LIN {X 0,Y 360.281,Z 704.675,A -85,B 0,C 180,E1 -13053.355,E2 -13053.355} C_VEL
LIN {X 0,Y 360.322,Z 702.646,A -85,B 0,C 180,E1 -13055.597,E2 -13055.597} C_VEL
LIN {X 0,Y 360.498,Z 699.39,A -85,B 0,C 180,E1 -13057.843,E2 -13057.843} C_VEL
LIN {X 0,Y 360.868,Z 694.879,A -85,B 0,C 180,E1 -13060.095,E2 -13060.095} C_VEL
LIN {X 0,Y 361.629,Z 689.019,A -85,B 0,C 180,E1 -13062.344,E2 -13062.344} C_VEL
LIN {X 0,Y 362.564,Z 681.663,A -85,B 0,C 180,E1 -13064.596,E2 -13064.596} C_VEL
LIN {X 0,Y 363.854,Z 673.825,A -85,B 0,C 180,E1 -13066.553,E2 -13066.553} C_VEL
LIN {X 0,Y 365.455,Z 664.444,A -85,B 0,C 180,E1 -13068.5,E2 -13068.5} C_VEL
LIN {X 0,Y 367.139,Z 654.928,A -85,B 0,C 180,E1 -13070.155,E2 -13070.155} C_VEL
LIN {X 0,Y 369.018,Z 643.667,A -85,B 0,C 180,E1 -13071.801,E2 -13071.801} C_VEL
LIN {X 0,Y 371.077,Z 631.324,A -85,B 0,C 180,E1 -13073.289,E2 -13073.289} C_VEL
LIN {X 0,Y 373.236,Z 617.701,A -85,B 0,C 180,E1 -13074.621,E2 -13074.621} C_VEL
LIN {X 0,Y 375.112,Z 604.087,A -85,B 0,C 180,E1 -13075.697,E2 -13075.697} C_VEL
LIN {X 0,Y 376.684,Z 589.68,A -85,B 0,C 180,E1 -13076.601,E2 -13076.601} C_VEL
LIN {X 0,Y 378.096,Z 575.109,A -85,B 0,C 180,E1 -13077.278,E2 -13077.278} C_VEL
LIN {X 0,Y 379.101,Z 560.278,A -85,B 0,C 180,E1 -13077.761,E2 -13077.761} C_VEL
LIN {X 0,Y 380.462,Z 514.951,A -85,B 0,C 180,E1 -13078.666,E2 -13078.666} C_VEL
LIN {X 0,Y 382.505,Z 436.101,A -85,B 0,C 180,E1 -13080.202,E2 -13080.202} C_VEL
LIN {X 0,Y 378.894,Z 417.126,A -85,B 0,C 180,E1 -13080.986,E2 -13080.986} C_VEL
LIN {X 0,Y 377.468,Z 411.276,A -85,B 0,C 180,E1 -13081.265,E2 -13081.265} C_VEL
LIN {X 0,Y 372.216,Z 400.047,A -85,B 0,C 180,E1 -13082.081,E2 -13082.081} C_VEL
LIN {X 0,Y 368.416,Z 392.244,A -85,B 0,C 180,E1 -13082.715,E2 -13082.715} C_VEL
LIN {X 0,Y 365.416,Z 380.947,A -85,B 0,C 180,E1 -13085.538,E2 -13085.538} C_VEL
LIN {X 0,Y 361.841,Z 369.028,A -85,B 0,C 180,E1 -13088.773,E2 -13088.773} C_VEL
LIN {X 0,Y 361.828,Z 369.03,A -85,B 0,C 180,E1 -13092.431,E2 -13092.431} C_VEL
LIN {X 0,Y 361.815,Z 369.04,A -85,B 0,C 180,E1 -13095.947,E2 -13095.947} C_VEL
LIN {X 0,Y 361.811,Z 369.041,A -85,B 0,C 180,E1 -13099.249,E2 -13099.249} C_VEL
LIN {X 0,Y 361.862,Z 369.019,A -85,B 0,C 180,E1 -13102.982,E2 -13102.982} C_VEL
LIN {X 0,Y 361.861,Z 369.033,A -85,B 0,C 180,E1 -13106.63,E2 -13106.63} C_VEL
LIN {X 0,Y 361.864,Z 369.009,A -85,B 0,C 180,E1 -13109.672,E2 -13109.672} C_VEL
LIN {X 0,Y 361.873,Z 369.027,A -85,B 0,C 180,E1 -13113.469,E2 -13113.469} C_VEL
LIN {X 0,Y 361.88,Z 369.026,A -85,B 0,C 180,E1 -13117.144,E2 -13117.144} C_VEL
LIN {X 0,Y 361.888,Z 369.027,A -85,B 0,C 180,E1 -13120.723,E2 -13120.723} C_VEL
LIN {X 0,Y 361.933,Z 369.022,A -85,B 0,C 180,E1 -13123.066,E2 -13123.066} C_VEL
LIN {X 0,Y 362,Z 369.016,A -85,B 0,C 180,E1 -13126.528,E2 -13126.528} C_VEL
LIN {X 0,Y 362.001,Z 369.018,A -85,B 0,C 180,E1 -13129.938,E2 -13129.938} C_VEL
LIN {X 0,Y 362.125,Z 369.001,A -85,B 0,C 180,E1 -13133.313,E2 -13133.313} C_VEL
LIN {X 0,Y 362.278,Z 368.982,A -85,B 0,C 180,E1 -13137.777,E2 -13137.777} C_VEL
LIN {X 0,Y 362.206,Z 368.992,A -85,B 0,C 180,E1 -13141.112,E2 -13141.112} C_VEL
LIN {X 0,Y 362.271,Z 368.984,A -85,B 0,C 180,E1 -13142.224,E2 -13142.224} C_VEL
LIN {X 0,Y 362.126,Z 368.996,A -85,B 0,C 180,E1 -13146.688,E2 -13146.688} C_VEL
LIN {X 0,Y 362.03,Z 369.014,A -85,B 0,C 180,E1 -13150.063,E2 -13150.063} C_VEL
LIN {X 0,Y 362,Z 369.017,A -85,B 0,C 180,E1 -13153.899,E2 -13153.899} C_VEL
LIN {X 0,Y 361.97,Z 369.011,A -85,B 0,C 180,E1 -13157.939,E2 -13157.939} C_VEL
LIN {X 0,Y 361.863,Z 369.029,A -85,B 0,C 180,E1 -13161.655,E2 -13161.655} C_VEL
LIN {X 0,Y 361.872,Z 369.011,A -85,B 0,C 180,E1 -13165.295,E2 -13165.295} C_VEL
LIN {X 0,Y 361.877,Z 369.03,A -85,B 0,C 180,E1 -13169.08,E2 -13169.08} C_VEL
LIN {X 0,Y 361.851,Z 369.038,A -85,B 0,C 180,E1 -13172.945,E2 -13172.945} C_VEL
LIN {X 0,Y 361.867,Z 369.018,A -85,B 0,C 180,E1 -13175.638,E2 -13175.638} C_VEL
LIN {X 0,Y 361.828,Z 369.028,A -85,B 0,C 180,E1 -13179.018,E2 -13179.018} C_VEL
LIN {X 0,Y 361.836,Z 369.03,A -85,B 0,C 180,E1 -13182.83,E2 -13182.83} C_VEL
LIN {X 0,Y 361.874,Z 369.139,A -85,B 0,C 180,E1 -13185.189,E2 -13185.189} C_VEL
LIN {X 0,Y 363.464,Z 374.54,A -85,B 0,C 180,E1 -13186.781,E2 -13186.781} C_VEL
LIN {X 0,Y 374.259,Z 394.401,A -85,B 0,C 180,E1 -13188.479,E2 -13188.479} C_VEL
LIN {X 0,Y 382.475,Z 411.542,A -85,B 0,C 180,E1 -13189.721,E2 -13189.721} C_VEL
LIN {X 0,Y 383.173,Z 413.081,A -85,B 0,C 180,E1 -13189.825,E2 -13189.825} C_VEL
LIN {X 0,Y 379.937,Z 522.43,A -85,B 0,C 180,E1 -13191.918,E2 -13191.918} C_VEL
LIN {X 0,Y 379.375,Z 541.692,A -85,B 0,C 180,E1 -13192.35,E2 -13192.35} C_VEL
LIN {X 0,Y 378.405,Z 556.889,A -85,B 0,C 180,E1 -13192.885,E2 -13192.885} C_VEL
LIN {X 0,Y 377.255,Z 570.714,A -85,B 0,C 180,E1 -13193.572,E2 -13193.572} C_VEL
LIN {X 0,Y 375.754,Z 583.754,A -85,B 0,C 180,E1 -13194.398,E2 -13194.398} C_VEL
LIN {X 0,Y 374.107,Z 597.673,A -85,B 0,C 180,E1 -13195.533,E2 -13195.533} C_VEL
LIN {X 0,Y 372.22,Z 610.378,A -85,B 0,C 180,E1 -13196.8,E2 -13196.8} C_VEL
LIN {X 0,Y 370.129,Z 623.095,A -85,B 0,C 180,E1 -13198.346,E2 -13198.346} C_VEL
LIN {X 0,Y 368.249,Z 633.861,A -85,B 0,C 180,E1 -13199.935,E2 -13199.935} C_VEL
LIN {X 0,Y 366.464,Z 644.127,A -85,B 0,C 180,E1 -13201.755,E2 -13201.755} C_VEL
LIN {X 0,Y 364.771,Z 653.232,A -85,B 0,C 180,E1 -13203.696,E2 -13203.696} C_VEL
LIN {X 0,Y 363.385,Z 660.855,A -85,B 0,C 180,E1 -13205.661,E2 -13205.661} C_VEL
LIN {X 0,Y 362.26,Z 667.561,A -85,B 0,C 180,E1 -13207.771,E2 -13207.771} C_VEL
LIN {X 0,Y 361.372,Z 673.427,A -85,B 0,C 180,E1 -13210.102,E2 -13210.102} C_VEL
LIN {X 0,Y 360.817,Z 678.163,A -85,B 0,C 180,E1 -13212.637,E2 -13212.637} C_VEL
LIN {X 0,Y 360.53,Z 680.275,A -85,B 0,C 180,E1 -13214.163,E2 -13214.163} C_VEL
LIN {X 0,Y 360.307,Z 682.413,A -85,B 0,C 180,E1 -13216.463,E2 -13216.463} C_VEL
LIN {X 0,Y 360.253,Z 683.361,A -85,B 0,C 180,E1 -13218.75,E2 -13218.75} C_VEL
LIN {X 0,Y 360.177,Z 683.159,A -85,B 0,C 180,E1 -13221.019,E2 -13221.019} C_VEL
LIN {X 0,Y 360.356,Z 681.807,A -85,B 0,C 180,E1 -13223.28,E2 -13223.28} C_VEL
LIN {X 0,Y 360.509,Z 679.255,A -85,B 0,C 180,E1 -13225.528,E2 -13225.528} C_VEL
LIN {X 0,Y 360.794,Z 675.491,A -85,B 0,C 180,E1 -13227.767,E2 -13227.767} C_VEL
LIN {X 0,Y 361.121,Z 670.466,A -85,B 0,C 180,E1 -13230,E2 -13230} C_VEL
LIN {X 0,Y 361.852,Z 664.03,A -85,B 0,C 180,E1 -13232.226,E2 -13232.226} C_VEL
LIN {X 0,Y 362.935,Z 655.999,A -85,B 0,C 180,E1 -13234.443,E2 -13234.443} C_VEL
LIN {X 0,Y 364.185,Z 647.445,A -85,B 0,C 180,E1 -13236.371,E2 -13236.371} C_VEL
LIN {X 0,Y 365.609,Z 637.19,A -85,B 0,C 180,E1 -13238.289,E2 -13238.289} C_VEL
LIN {X 0,Y 367.078,Z 626.692,A -85,B 0,C 180,E1 -13239.922,E2 -13239.922} C_VEL
LIN {X 0,Y 368.588,Z 615.282,A -85,B 0,C 180,E1 -13241.41,E2 -13241.41} C_VEL
LIN {X 0,Y 370.142,Z 602.884,A -85,B 0,C 180,E1 -13242.752,E2 -13242.752} C_VEL
LIN {X 0,Y 371.609,Z 590.122,A -85,B 0,C 180,E1 -13243.886,E2 -13243.886} C_VEL
LIN {X 0,Y 371.551,Z 584.912,A -85,B 0,C 180,E1 -13244.323,E2 -13244.323} C_VEL
LIN {X 0,Y 369.644,Z 576.463,A -85,B 0,C 180,E1 -13245.078,E2 -13245.078} C_VEL
LIN {X 0,Y 367.665,Z 567.83,A -85,B 0,C 180,E1 -13245.765,E2 -13245.765} C_VEL
LIN {X 0,Y 367.506,Z 562.338,A -85,B 0,C 180,E1 -13246.09,E2 -13246.09} C_VEL
LIN {X 0,Y 368.412,Z 546.776,A -85,B 0,C 180,E1 -13246.735,E2 -13246.735} C_VEL
LIN {X 0,Y 369.037,Z 531.674,A -85,B 0,C 180,E1 -13247.133,E2 -13247.133} C_VEL
LIN {X 0,Y 371.931,Z 411.976,A -85,B 0,C 180,E1 -13249.45,E2 -13249.45} C_VEL
LIN {X 0,Y 369.611,Z 405.572,A -85,B 0,C 180,E1 -13249.766,E2 -13249.766} C_VEL
LIN {X 0,Y 360.274,Z 383.68,A -85,B 0,C 180,E1 -13251,E2 -13251} C_VEL
LIN {X 0,Y 355.812,Z 373.961,A -85,B 0,C 180,E1 -13251.636,E2 -13251.636} C_VEL
LIN {X 0,Y 354.836,Z 369.91,A -85,B 0,C 180,E1 -13252.72,E2 -13252.72} C_VEL
LIN {X 0,Y 354.807,Z 369.916,A -85,B 0,C 180,E1 -13255.835,E2 -13255.835} C_VEL
LIN {X 0,Y 354.804,Z 369.909,A -85,B 0,C 180,E1 -13259.683,E2 -13259.683} C_VEL
LIN {X 0,Y 354.791,Z 369.907,A -85,B 0,C 180,E1 -13262.333,E2 -13262.333} C_VEL
LIN {X 0,Y 354.825,Z 369.904,A -85,B 0,C 180,E1 -13265.699,E2 -13265.699} C_VEL
LIN {X 0,Y 354.772,Z 369.913,A -85,B 0,C 180,E1 -13269.412,E2 -13269.412} C_VEL
LIN {X 0,Y 354.789,Z 369.914,A -85,B 0,C 180,E1 -13272.866,E2 -13272.866} C_VEL
LIN {X 0,Y 354.769,Z 369.902,A -85,B 0,C 180,E1 -13276.103,E2 -13276.103} C_VEL
LIN {X 0,Y 354.769,Z 369.919,A -85,B 0,C 180,E1 -13279.176,E2 -13279.176} C_VEL
LIN {X 0,Y 354.802,Z 369.912,A -85,B 0,C 180,E1 -13282.404,E2 -13282.404} C_VEL
LIN {X 0,Y 354.811,Z 369.911,A -85,B 0,C 180,E1 -13284.94,E2 -13284.94} C_VEL
LIN {X 0,Y 354.796,Z 369.915,A -85,B 0,C 180,E1 -13288.405,E2 -13288.405} C_VEL
LIN {X 0,Y 354.8,Z 369.891,A -85,B 0,C 180,E1 -13291.614,E2 -13291.614} C_VEL
LIN {X 0,Y 354.806,Z 369.882,A -85,B 0,C 180,E1 -13295.419,E2 -13295.419} C_VEL
LIN {X 0,Y 354.83,Z 369.91,A -85,B 0,C 180,E1 -13299.113,E2 -13299.113} C_VEL
LIN {X 0,Y 354.883,Z 369.889,A -85,B 0,C 180,E1 -13302.719,E2 -13302.719} C_VEL
LIN {X 0,Y 354.954,Z 369.891,A -85,B 0,C 180,E1 -13306.255,E2 -13306.255} C_VEL
LIN {X 0,Y 354.958,Z 369.885,A -85,B 0,C 180,E1 -13309.735,E2 -13309.735} C_VEL
LIN {X 0,Y 355.088,Z 369.876,A -85,B 0,C 180,E1 -13313.179,E2 -13313.179} C_VEL
LIN {X 0,Y 355.229,Z 369.862,A -85,B 0,C 180,E1 -13317.732,E2 -13317.732} C_VEL
LIN {X 0,Y 355.149,Z 369.859,A -85,B 0,C 180,E1 -13321.133,E2 -13321.133} C_VEL
LIN {X 0,Y 355.236,Z 369.85,A -85,B 0,C 180,E1 -13322.267,E2 -13322.267} C_VEL
LIN {X 0,Y 355.09,Z 369.872,A -85,B 0,C 180,E1 -13326.82,E2 -13326.82} C_VEL
LIN {X 0,Y 354.958,Z 369.892,A -85,B 0,C 180,E1 -13330.264,E2 -13330.264} C_VEL
LIN {X 0,Y 354.925,Z 369.893,A -85,B 0,C 180,E1 -13334.006,E2 -13334.006} C_VEL
LIN {X 0,Y 354.891,Z 369.894,A -85,B 0,C 180,E1 -13338.091,E2 -13338.091} C_VEL
LIN {X 0,Y 354.831,Z 369.901,A -85,B 0,C 180,E1 -13342.106,E2 -13342.106} C_VEL
LIN {X 0,Y 354.814,Z 369.907,A -85,B 0,C 180,E1 -13345.834,E2 -13345.834} C_VEL
LIN {X 0,Y 354.799,Z 369.912,A -85,B 0,C 180,E1 -13349.683,E2 -13349.683} C_VEL
LIN {X 0,Y 354.787,Z 369.912,A -85,B 0,C 180,E1 -13352.333,E2 -13352.333} C_VEL
LIN {X 0,Y 354.821,Z 369.91,A -85,B 0,C 180,E1 -13355.699,E2 -13355.699} C_VEL
LIN {X 0,Y 354.767,Z 369.907,A -85,B 0,C 180,E1 -13359.412,E2 -13359.412} C_VEL
LIN {X 0,Y 354.784,Z 369.914,A -85,B 0,C 180,E1 -13362.866,E2 -13362.866} C_VEL
LIN {X 0,Y 354.765,Z 369.92,A -85,B 0,C 180,E1 -13366.103,E2 -13366.103} C_VEL
LIN {X 0,Y 354.764,Z 369.919,A -85,B 0,C 180,E1 -13369.176,E2 -13369.176} C_VEL
LIN {X 0,Y 354.799,Z 369.914,A -85,B 0,C 180,E1 -13372.404,E2 -13372.404} C_VEL
LIN {X 0,Y 354.847,Z 369.999,A -85,B 0,C 180,E1 -13373.576,E2 -13373.576} C_VEL
LIN {X 0,Y 357.911,Z 382.015,A -85,B 0,C 180,E1 -13376.4,E2 -13376.4} C_VEL
LIN {X 0,Y 360.445,Z 392.787,A -85,B 0,C 180,E1 -13378.815,E2 -13378.815} C_VEL
LIN {X 0,Y 366.239,Z 407.269,A -85,B 0,C 180,E1 -13379.603,E2 -13379.603} C_VEL
LIN {X 0,Y 371.489,Z 436.998,A -85,B 0,C 180,E1 -13380.645,E2 -13380.645} C_VEL
LIN {X 0,Y 368.547,Z 559.048,A -85,B 0,C 180,E1 -13383.032,E2 -13383.032} C_VEL
LIN {X 0,Y 367.718,Z 573.654,A -85,B 0,C 180,E1 -13383.502,E2 -13383.502} C_VEL
LIN {X 0,Y 366.531,Z 587.928,A -85,B 0,C 180,E1 -13384.157,E2 -13384.157} C_VEL
LIN {X 0,Y 365.204,Z 602.116,A -85,B 0,C 180,E1 -13385.028,E2 -13385.028} C_VEL
LIN {X 0,Y 363.669,Z 615.368,A -85,B 0,C 180,E1 -13386.057,E2 -13386.057} C_VEL
LIN {X 0,Y 362.049,Z 628.373,A -85,B 0,C 180,E1 -13387.306,E2 -13387.306} C_VEL
LIN {X 0,Y 360.326,Z 640.376,A -85,B 0,C 180,E1 -13388.699,E2 -13388.699} C_VEL
LIN {X 0,Y 358.764,Z 652.106,A -85,B 0,C 180,E1 -13390.348,E2 -13390.348} C_VEL
LIN {X 0,Y 357.427,Z 661.768,A -85,B 0,C 180,E1 -13391.959,E2 -13391.959} C_VEL
LIN {X 0,Y 356.022,Z 671.76,A -85,B 0,C 180,E1 -13393.957,E2 -13393.957} C_VEL
LIN {X 0,Y 354.962,Z 680.097,A -85,B 0,C 180,E1 -13395.968,E2 -13395.968} C_VEL
LIN {X 0,Y 354.234,Z 686.934,A -85,B 0,C 180,E1 -13397.976,E2 -13397.976} C_VEL
LIN {X 0,Y 353.629,Z 693.271,A -85,B 0,C 180,E1 -13400.274,E2 -13400.274} C_VEL
LIN {X 0,Y 353.371,Z 698.169,A -85,B 0,C 180,E1 -13402.572,E2 -13402.572} C_VEL
LIN {X 0,Y 353.259,Z 701.01,A -85,B 0,C 180,E1 -13404.291,E2 -13404.291} C_VEL
LIN {X 0,Y 353.209,Z 703.639,A -85,B 0,C 180,E1 -13406.578,E2 -13406.578} C_VEL
LIN {X 0,Y 353.241,Z 705.069,A -85,B 0,C 180,E1 -13408.86,E2 -13408.86} C_VEL
LIN {X 0,Y 353.235,Z 705.351,A -85,B 0,C 180,E1 -13411.14,E2 -13411.14} C_VEL
LIN {X 0,Y 353.201,Z 704.496,A -85,B 0,C 180,E1 -13413.422,E2 -13413.422} C_VEL
LIN {X 0,Y 353.275,Z 702.246,A -85,B 0,C 180,E1 -13415.908,E2 -13415.908} C_VEL
LIN {X 0,Y 353.506,Z 698.259,A -85,B 0,C 180,E1 -13418.575,E2 -13418.575} C_VEL
LIN {X 0,Y 353.959,Z 693.486,A -85,B 0,C 180,E1 -13420.873,E2 -13420.873} C_VEL
LIN {X 0,Y 354.8,Z 687.326,A -85,B 0,C 180,E1 -13423.167,E2 -13423.167} C_VEL
LIN {X 0,Y 356.02,Z 679.611,A -85,B 0,C 180,E1 -13425.456,E2 -13425.456} C_VEL
LIN {X 0,Y 357.44,Z 671.406,A -85,B 0,C 180,E1 -13427.448,E2 -13427.448} C_VEL
LIN {X 0,Y 359.305,Z 661.575,A -85,B 0,C 180,E1 -13429.422,E2 -13429.422} C_VEL
LIN {X 0,Y 361.368,Z 649.929,A -85,B 0,C 180,E1 -13431.357,E2 -13431.357} C_VEL
LIN {X 0,Y 363.585,Z 637.487,A -85,B 0,C 180,E1 -13433.043,E2 -13433.043} C_VEL
LIN {X 0,Y 365.692,Z 625.242,A -85,B 0,C 180,E1 -13434.406,E2 -13434.406} C_VEL
LIN {X 0,Y 367.733,Z 611.898,A -85,B 0,C 180,E1 -13435.62,E2 -13435.62} C_VEL
LIN {X 0,Y 369.551,Z 597.796,A -85,B 0,C 180,E1 -13436.651,E2 -13436.651} C_VEL
LIN {X 0,Y 371.181,Z 582.922,A -85,B 0,C 180,E1 -13437.485,E2 -13437.485} C_VEL
LIN {X 0,Y 372.544,Z 567.562,A -85,B 0,C 180,E1 -13438.101,E2 -13438.101} C_VEL
LIN {X 0,Y 373.45,Z 551.16,A -85,B 0,C 180,E1 -13438.525,E2 -13438.525} C_VEL
LIN {X 0,Y 376.625,Z 438.24,A -85,B 0,C 180,E1 -13440.741,E2 -13440.741} C_VEL
LIN {X 0,Y 373.655,Z 421.477,A -85,B 0,C 180,E1 -13441.431,E2 -13441.431} C_VEL
LIN {X 0,Y 371.998,Z 414.427,A -85,B 0,C 180,E1 -13441.771,E2 -13441.771} C_VEL
LIN {X 0,Y 366.809,Z 403.301,A -85,B 0,C 180,E1 -13442.602,E2 -13442.602} C_VEL
LIN {X 0,Y 361.173,Z 391.955,A -85,B 0,C 180,E1 -13443.563,E2 -13443.563} C_VEL
LIN {X 0,Y 358.117,Z 380.966,A -85,B 0,C 180,E1 -13446.427,E2 -13446.427} C_VEL
LIN {X 0,Y 355.208,Z 371.575,A -85,B 0,C 180,E1 -13449.052,E2 -13449.052} C_VEL
LIN {X 0,Y 354.771,Z 369.91,A -85,B 0,C 180,E1 -13449.555,E2 -13449.555} C_VEL
LIN {X 0,Y 354.784,Z 369.911,A -85,B 0,C 180,E1 -13452.867,E2 -13452.867} C_VEL
LIN {X 0,Y 354.764,Z 369.918,A -85,B 0,C 180,E1 -13456.104,E2 -13456.104} C_VEL
LIN {X 0,Y 354.764,Z 369.919,A -85,B 0,C 180,E1 -13459.176,E2 -13459.176} C_VEL
LIN {X 0,Y 354.799,Z 369.905,A -85,B 0,C 180,E1 -13462.405,E2 -13462.405} C_VEL
LIN {X 0,Y 354.811,Z 369.9,A -85,B 0,C 180,E1 -13464.941,E2 -13464.941} C_VEL
LIN {X 0,Y 354.794,Z 369.892,A -85,B 0,C 180,E1 -13468.405,E2 -13468.405} C_VEL
LIN {X 0,Y 354.802,Z 369.911,A -85,B 0,C 180,E1 -13471.615,E2 -13471.615} C_VEL
LIN {X 0,Y 354.85,Z 369.907,A -85,B 0,C 180,E1 -13475.423,E2 -13475.423} C_VEL
LIN {X 0,Y 354.84,Z 369.908,A -85,B 0,C 180,E1 -13479.114,E2 -13479.114} C_VEL
LIN {X 0,Y 354.899,Z 369.901,A -85,B 0,C 180,E1 -13482.72,E2 -13482.72} C_VEL
LIN {X 0,Y 354.953,Z 369.898,A -85,B 0,C 180,E1 -13486.256,E2 -13486.256} C_VEL
LIN {X 0,Y 354.957,Z 369.894,A -85,B 0,C 180,E1 -13489.736,E2 -13489.736} C_VEL
LIN {X 0,Y 355.09,Z 369.878,A -85,B 0,C 180,E1 -13493.18,E2 -13493.18} C_VEL
LIN {X 0,Y 355.241,Z 369.859,A -85,B 0,C 180,E1 -13497.733,E2 -13497.733} C_VEL
LIN {X 0,Y 355.174,Z 369.867,A -85,B 0,C 180,E1 -13501.134,E2 -13501.134} C_VEL
LIN {X 0,Y 355.233,Z 369.86,A -85,B 0,C 180,E1 -13502.268,E2 -13502.268} C_VEL
LIN {X 0,Y 355.091,Z 369.871,A -85,B 0,C 180,E1 -13506.821,E2 -13506.821} C_VEL
LIN {X 0,Y 354.978,Z 369.89,A -85,B 0,C 180,E1 -13510.265,E2 -13510.265} C_VEL
LIN {X 0,Y 354.945,Z 369.894,A -85,B 0,C 180,E1 -13514.019,E2 -13514.019} C_VEL
LIN {X 0,Y 354.925,Z 369.885,A -85,B 0,C 180,E1 -13518.109,E2 -13518.109} C_VEL
LIN {X 0,Y 354.817,Z 369.909,A -85,B 0,C 180,E1 -13522.108,E2 -13522.108} C_VEL
LIN {X 0,Y 354.816,Z 369.888,A -85,B 0,C 180,E1 -13525.835,E2 -13525.835} C_VEL
LIN {X 0,Y 354.81,Z 369.906,A -85,B 0,C 180,E1 -13529.683,E2 -13529.683} C_VEL
LIN {X 0,Y 354.817,Z 369.913,A -85,B 0,C 180,E1 -13533.684,E2 -13533.684} C_VEL
LIN {X 0,Y 354.795,Z 369.905,A -85,B 0,C 180,E1 -13536.461,E2 -13536.461} C_VEL
LIN {X 0,Y 354.771,Z 369.906,A -85,B 0,C 180,E1 -13539.413,E2 -13539.413} C_VEL
LIN {X 0,Y 354.788,Z 369.908,A -85,B 0,C 180,E1 -13542.867,E2 -13542.867} C_VEL
LIN {X 0,Y 354.791,Z 369.931,A -85,B 0,C 180,E1 -13544.415,E2 -13544.415} C_VEL
LIN {X 0,Y 356.258,Z 374.894,A -85,B 0,C 180,E1 -13545.92,E2 -13545.92} C_VEL
LIN {X 0,Y 367.693,Z 395.463,A -85,B 0,C 180,E1 -13547.781,E2 -13547.781} C_VEL
LIN {X 0,Y 375.566,Z 411.574,A -85,B 0,C 180,E1 -13549.013,E2 -13549.013} C_VEL
LIN {X 0,Y 377.203,Z 415.21,A -85,B 0,C 180,E1 -13549.267,E2 -13549.267} C_VEL
LIN {X 0,Y 374.022,Z 519.338,A -85,B 0,C 180,E1 -13551.291,E2 -13551.291} C_VEL
LIN {X 0,Y 373.33,Z 541.069,A -85,B 0,C 180,E1 -13551.764,E2 -13551.764} C_VEL
LIN {X 0,Y 372.344,Z 556.014,A -85,B 0,C 180,E1 -13552.28,E2 -13552.28} C_VEL
LIN {X 0,Y 371.092,Z 571.056,A -85,B 0,C 180,E1 -13553.037,E2 -13553.037} C_VEL
LIN {X 0,Y 369.528,Z 584.075,A -85,B 0,C 180,E1 -13553.872,E2 -13553.872} C_VEL
LIN {X 0,Y 367.817,Z 597.97,A -85,B 0,C 180,E1 -13555.025,E2 -13555.025} C_VEL
LIN {X 0,Y 365.838,Z 610.651,A -85,B 0,C 180,E1 -13556.309,E2 -13556.309} C_VEL
LIN {X 0,Y 363.61,Z 623.459,A -85,B 0,C 180,E1 -13557.892,E2 -13557.892} C_VEL
LIN {X 0,Y 361.503,Z 635.013,A -85,B 0,C 180,E1 -13559.638,E2 -13559.638} C_VEL
LIN {X 0,Y 359.54,Z 645.676,A -85,B 0,C 180,E1 -13561.599,E2 -13561.599} C_VEL
LIN {X 0,Y 357.887,Z 654.098,A -85,B 0,C 180,E1 -13563.464,E2 -13563.464} C_VEL
LIN {X 0,Y 356.394,Z 661.85,A -85,B 0,C 180,E1 -13565.536,E2 -13565.536} C_VEL
LIN {X 0,Y 355.117,Z 669.027,A -85,B 0,C 180,E1 -13567.912,E2 -13567.912} C_VEL
LIN {X 0,Y 354.248,Z 674.601,A -85,B 0,C 180,E1 -13570.29,E2 -13570.29} C_VEL
LIN {X 0,Y 353.734,Z 678.741,A -85,B 0,C 180,E1 -13572.661,E2 -13572.661} C_VEL
LIN {X 0,Y 353.335,Z 681.577,A -85,B 0,C 180,E1 -13575.014,E2 -13575.014} C_VEL
LIN {X 0,Y 353.249,Z 683.193,A -85,B 0,C 180,E1 -13577.359,E2 -13577.359} C_VEL
LIN {X 0,Y 353.074,Z 683.645,A -85,B 0,C 180,E1 -13579.68,E2 -13579.68} C_VEL
LIN {X 0,Y 353.148,Z 682.942,A -85,B 0,C 180,E1 -13581.992,E2 -13581.992} C_VEL
LIN {X 0,Y 353.341,Z 681.04,A -85,B 0,C 180,E1 -13584.293,E2 -13584.293} C_VEL
LIN {X 0,Y 353.485,Z 677.969,A -85,B 0,C 180,E1 -13586.581,E2 -13586.581} C_VEL
LIN {X 0,Y 353.828,Z 673.667,A -85,B 0,C 180,E1 -13588.862,E2 -13588.862} C_VEL
LIN {X 0,Y 354.36,Z 668.045,A -85,B 0,C 180,E1 -13591.136,E2 -13591.136} C_VEL
LIN {X 0,Y 355.3,Z 660.934,A -85,B 0,C 180,E1 -13593.402,E2 -13593.402} C_VEL
LIN {X 0,Y 356.426,Z 653.333,A -85,B 0,C 180,E1 -13595.374,E2 -13595.374} C_VEL
LIN {X 0,Y 357.739,Z 644.221,A -85,B 0,C 180,E1 -13597.337,E2 -13597.337} C_VEL
LIN {X 0,Y 359.109,Z 634.975,A -85,B 0,C 180,E1 -13599.008,E2 -13599.008} C_VEL
LIN {X 0,Y 360.906,Z 622.989,A -85,B 0,C 180,E1 -13600.803,E2 -13600.803} C_VEL
LIN {X 0,Y 362.492,Z 610.817,A -85,B 0,C 180,E1 -13602.314,E2 -13602.314} C_VEL
LIN {X 0,Y 364.141,Z 597.407,A -85,B 0,C 180,E1 -13603.676,E2 -13603.676} C_VEL
LIN {X 0,Y 365.557,Z 584.26,A -85,B 0,C 180,E1 -13604.758,E2 -13604.758} C_VEL
LIN {X 0,Y 366.908,Z 569.786,A -85,B 0,C 180,E1 -13605.698,E2 -13605.698} C_VEL
LIN {X 0,Y 367.506,Z 562.338,A -85,B 0,C 180,E1 -13606.09,E2 -13606.09} C_VEL
LIN {X 0,Y 367.409,Z 556.765,A -85,B 0,C 180,E1 -13606.39,E2 -13606.39} C_VEL
LIN {X 0,Y 365.271,Z 547.698,A -85,B 0,C 180,E1 -13606.922,E2 -13606.922} C_VEL
LIN {X 0,Y 362.974,Z 538.503,A -85,B 0,C 180,E1 -13607.389,E2 -13607.389} C_VEL
LIN {X 0,Y 362.535,Z 532.726,A -85,B 0,C 180,E1 -13607.567,E2 -13607.567} C_VEL
LIN {X 0,Y 365.518,Z 413.122,A -85,B 0,C 180,E1 -13609.925,E2 -13609.925} C_VEL
LIN {X 0,Y 356.043,Z 390.405,A -85,B 0,C 180,E1 -13611.208,E2 -13611.208} C_VEL
LIN {X 0,Y 348.664,Z 374.277,A -85,B 0,C 180,E1 -13612.248,E2 -13612.248} C_VEL
LIN {X 0,Y 347.791,Z 370.787,A -85,B 0,C 180,E1 -13613.207,E2 -13613.207} C_VEL
LIN {X 0,Y 347.76,Z 370.793,A -85,B 0,C 180,E1 -13617.224,E2 -13617.224} C_VEL
LIN {X 0,Y 347.745,Z 370.791,A -85,B 0,C 180,E1 -13620.348,E2 -13620.348} C_VEL
LIN {X 0,Y 347.753,Z 370.793,A -85,B 0,C 180,E1 -13624.044,E2 -13624.044} C_VEL
LIN {X 0,Y 347.759,Z 370.786,A -85,B 0,C 180,E1 -13627.321,E2 -13627.321} C_VEL
LIN {X 0,Y 347.745,Z 370.784,A -85,B 0,C 180,E1 -13631.601,E2 -13631.601} C_VEL
LIN {X 0,Y 347.708,Z 370.788,A -85,B 0,C 180,E1 -13635.027,E2 -13635.027} C_VEL
LIN {X 0,Y 347.745,Z 370.791,A -85,B 0,C 180,E1 -13638.399,E2 -13638.399} C_VEL
LIN {X 0,Y 347.758,Z 370.789,A -85,B 0,C 180,E1 -13642.678,E2 -13642.678} C_VEL
LIN {X 0,Y 347.751,Z 370.786,A -85,B 0,C 180,E1 -13645.956,E2 -13645.956} C_VEL
LIN {X 0,Y 347.741,Z 370.791,A -85,B 0,C 180,E1 -13649.651,E2 -13649.651} C_VEL
LIN {X 0,Y 347.737,Z 370.749,A -85,B 0,C 180,E1 -13653.599,E2 -13653.599} C_VEL
LIN {X 0,Y 347.755,Z 370.771,A -85,B 0,C 180,E1 -13656.159,E2 -13656.159} C_VEL
LIN {X 0,Y 347.803,Z 370.785,A -85,B 0,C 180,E1 -13659.908,E2 -13659.908} C_VEL
LIN {X 0,Y 347.835,Z 370.773,A -85,B 0,C 180,E1 -13663.568,E2 -13663.568} C_VEL
LIN {X 0,Y 347.892,Z 370.77,A -85,B 0,C 180,E1 -13667.16,E2 -13667.16} C_VEL
LIN {X 0,Y 347.937,Z 370.763,A -85,B 0,C 180,E1 -13670.7,E2 -13670.7} C_VEL
LIN {X 0,Y 348.04,Z 370.742,A -85,B 0,C 180,E1 -13674.205,E2 -13674.205} C_VEL
LIN {X 0,Y 348.191,Z 370.738,A -85,B 0,C 180,E1 -13677.686,E2 -13677.686} C_VEL
LIN {X 0,Y 348.12,Z 370.734,A -85,B 0,C 180,E1 -13681.156,E2 -13681.156} C_VEL
LIN {X 0,Y 348.197,Z 370.727,A -85,B 0,C 180,E1 -13682.313,E2 -13682.313} C_VEL
LIN {X 0,Y 348.057,Z 370.749,A -85,B 0,C 180,E1 -13686.958,E2 -13686.958} C_VEL
LIN {X 0,Y 347.898,Z 370.771,A -85,B 0,C 180,E1 -13690.475,E2 -13690.475} C_VEL
LIN {X 0,Y 347.881,Z 370.771,A -85,B 0,C 180,E1 -13694.137,E2 -13694.137} C_VEL
LIN {X 0,Y 347.83,Z 370.773,A -85,B 0,C 180,E1 -13698.258,E2 -13698.258} C_VEL
LIN {X 0,Y 347.787,Z 370.781,A -85,B 0,C 180,E1 -13701.634,E2 -13701.634} C_VEL
LIN {X 0,Y 347.769,Z 370.788,A -85,B 0,C 180,E1 -13705.111,E2 -13705.111} C_VEL
LIN {X 0,Y 347.736,Z 370.795,A -85,B 0,C 180,E1 -13707.7,E2 -13707.7} C_VEL
LIN {X 0,Y 347.741,Z 370.791,A -85,B 0,C 180,E1 -13710.348,E2 -13710.348} C_VEL
LIN {X 0,Y 347.748,Z 370.794,A -85,B 0,C 180,E1 -13714.043,E2 -13714.043} C_VEL
LIN {X 0,Y 347.755,Z 370.793,A -85,B 0,C 180,E1 -13717.321,E2 -13717.321} C_VEL
LIN {X 0,Y 347.74,Z 370.796,A -85,B 0,C 180,E1 -13721.601,E2 -13721.601} C_VEL
LIN {X 0,Y 347.703,Z 370.798,A -85,B 0,C 180,E1 -13725.027,E2 -13725.027} C_VEL
LIN {X 0,Y 347.74,Z 370.797,A -85,B 0,C 180,E1 -13728.399,E2 -13728.399} C_VEL
LIN {X 0,Y 347.763,Z 370.792,A -85,B 0,C 180,E1 -13732.679,E2 -13732.679} C_VEL
LIN {X 0,Y 347.782,Z 370.924,A -85,B 0,C 180,E1 -13733.076,E2 -13733.076} C_VEL
LIN {X 0,Y 350.803,Z 382.506,A -85,B 0,C 180,E1 -13735.878,E2 -13735.878} C_VEL
LIN {X 0,Y 353.232,Z 392.712,A -85,B 0,C 180,E1 -13738.199,E2 -13738.199} C_VEL
LIN {X 0,Y 360.136,Z 409.785,A -85,B 0,C 180,E1 -13739.165,E2 -13739.165} C_VEL
LIN {X 0,Y 365.077,Z 438.588,A -85,B 0,C 180,E1 -13740.189,E2 -13740.189} C_VEL
LIN {X 0,Y 362.047,Z 559.128,A -85,B 0,C 180,E1 -13742.585,E2 -13742.585} C_VEL
LIN {X 0,Y 361.143,Z 574.553,A -85,B 0,C 180,E1 -13743.099,E2 -13743.099} C_VEL
LIN {X 0,Y 359.906,Z 588.636,A -85,B 0,C 180,E1 -13743.769,E2 -13743.769} C_VEL
LIN {X 0,Y 358.508,Z 603.033,A -85,B 0,C 180,E1 -13744.684,E2 -13744.684} C_VEL
LIN {X 0,Y 356.924,Z 616.058,A -85,B 0,C 180,E1 -13745.73,E2 -13745.73} C_VEL
LIN {X 0,Y 355.239,Z 628.895,A -85,B 0,C 180,E1 -13747,E2 -13747} C_VEL
LIN {X 0,Y 353.469,Z 640.771,A -85,B 0,C 180,E1 -13748.418,E2 -13748.418} C_VEL
LIN {X 0,Y 351.813,Z 652.709,A -85,B 0,C 180,E1 -13750.147,E2 -13750.147} C_VEL
LIN {X 0,Y 350.341,Z 662.729,A -85,B 0,C 180,E1 -13751.884,E2 -13751.884} C_VEL
LIN {X 0,Y 348.938,Z 672.522,A -85,B 0,C 180,E1 -13753.922,E2 -13753.922} C_VEL
LIN {X 0,Y 347.849,Z 680.672,A -85,B 0,C 180,E1 -13755.969,E2 -13755.969} C_VEL
LIN {X 0,Y 347.021,Z 688.262,A -85,B 0,C 180,E1 -13758.315,E2 -13758.315} C_VEL
LIN {X 0,Y 346.501,Z 694.278,A -85,B 0,C 180,E1 -13760.662,E2 -13760.662} C_VEL
LIN {X 0,Y 346.237,Z 698.895,A -85,B 0,C 180,E1 -13763.005,E2 -13763.005} C_VEL
LIN {X 0,Y 346.142,Z 702.188,A -85,B 0,C 180,E1 -13765.341,E2 -13765.341} C_VEL
LIN {X 0,Y 346.107,Z 704.238,A -85,B 0,C 180,E1 -13767.672,E2 -13767.672} C_VEL
LIN {X 0,Y 346.18,Z 705.126,A -85,B 0,C 180,E1 -13770,E2 -13770} C_VEL
LIN {X 0,Y 346.092,Z 704.87,A -85,B 0,C 180,E1 -13772.328,E2 -13772.328} C_VEL
LIN {X 0,Y 346.121,Z 703.481,A -85,B 0,C 180,E1 -13774.659,E2 -13774.659} C_VEL
LIN {X 0,Y 346.226,Z 700.885,A -85,B 0,C 180,E1 -13776.996,E2 -13776.996} C_VEL
LIN {X 0,Y 346.562,Z 697.077,A -85,B 0,C 180,E1 -13779.337,E2 -13779.337} C_VEL
LIN {X 0,Y 347.182,Z 691.985,A -85,B 0,C 180,E1 -13781.679,E2 -13781.679} C_VEL
LIN {X 0,Y 348.077,Z 685.483,A -85,B 0,C 180,E1 -13784.022,E2 -13784.022} C_VEL
LIN {X 0,Y 349.517,Z 677.395,A -85,B 0,C 180,E1 -13786.35,E2 -13786.35} C_VEL
LIN {X 0,Y 351.101,Z 668.812,A -85,B 0,C 180,E1 -13788.377,E2 -13788.377} C_VEL
LIN {X 0,Y 353.093,Z 658.931,A -85,B 0,C 180,E1 -13790.308,E2 -13790.308} C_VEL
LIN {X 0,Y 355.094,Z 648.021,A -85,B 0,C 180,E1 -13792.089,E2 -13792.089} C_VEL
LIN {X 0,Y 357.259,Z 636.632,A -85,B 0,C 180,E1 -13793.629,E2 -13793.629} C_VEL
LIN {X 0,Y 359.478,Z 624.279,A -85,B 0,C 180,E1 -13795.01,E2 -13795.01} C_VEL
LIN {X 0,Y 361.612,Z 610.789,A -85,B 0,C 180,E1 -13796.241,E2 -13796.241} C_VEL
LIN {X 0,Y 363.575,Z 596.227,A -85,B 0,C 180,E1 -13797.297,E2 -13797.297} C_VEL
LIN {X 0,Y 365.242,Z 581.197,A -85,B 0,C 180,E1 -13798.127,E2 -13798.127} C_VEL
LIN {X 0,Y 366.581,Z 566.192,A -85,B 0,C 180,E1 -13798.718,E2 -13798.718} C_VEL
LIN {X 0,Y 367.417,Z 550.638,A -85,B 0,C 180,E1 -13799.116,E2 -13799.116} C_VEL
LIN {X 0,Y 370.73,Z 439.308,A -85,B 0,C 180,E1 -13801.33,E2 -13801.33} C_VEL
LIN {X 0,Y 367.735,Z 422.641,A -85,B 0,C 180,E1 -13802.042,E2 -13802.042} C_VEL
LIN {X 0,Y 366.451,Z 417.304,A -85,B 0,C 180,E1 -13802.31,E2 -13802.31} C_VEL
LIN {X 0,Y 360.347,Z 404.379,A -85,B 0,C 180,E1 -13803.322,E2 -13803.322} C_VEL
LIN {X 0,Y 353.912,Z 391.779,A -85,B 0,C 180,E1 -13804.433,E2 -13804.433} C_VEL
LIN {X 0,Y 350.582,Z 379.941,A -85,B 0,C 180,E1 -13807.643,E2 -13807.643} C_VEL
LIN {X 0,Y 347.735,Z 370.796,A -85,B 0,C 180,E1 -13810.392,E2 -13810.392} C_VEL
LIN {X 0,Y 347.721,Z 370.797,A -85,B 0,C 180,E1 -13813.409,E2 -13813.409} C_VEL
LIN {X 0,Y 347.723,Z 370.796,A -85,B 0,C 180,E1 -13816.687,E2 -13816.687} C_VEL
LIN {X 0,Y 347.7,Z 370.797,A -85,B 0,C 180,E1 -13820.183,E2 -13820.183} C_VEL
LIN {X 0,Y 347.755,Z 370.779,A -85,B 0,C 180,E1 -13822.679,E2 -13822.679} C_VEL
LIN {X 0,Y 347.748,Z 370.79,A -85,B 0,C 180,E1 -13825.957,E2 -13825.957} C_VEL
LIN {X 0,Y 347.74,Z 370.767,A -85,B 0,C 180,E1 -13829.652,E2 -13829.652} C_VEL
LIN {X 0,Y 347.755,Z 370.785,A -85,B 0,C 180,E1 -13833.602,E2 -13833.602} C_VEL
LIN {X 0,Y 347.771,Z 370.788,A -85,B 0,C 180,E1 -13836.161,E2 -13836.161} C_VEL
LIN {X 0,Y 347.806,Z 370.782,A -85,B 0,C 180,E1 -13839.909,E2 -13839.909} C_VEL
LIN {X 0,Y 347.867,Z 370.781,A -85,B 0,C 180,E1 -13842.36,E2 -13842.36} C_VEL
LIN {X 0,Y 347.898,Z 370.774,A -85,B 0,C 180,E1 -13845.971,E2 -13845.971} C_VEL
LIN {X 0,Y 347.897,Z 370.773,A -85,B 0,C 180,E1 -13849.525,E2 -13849.525} C_VEL
LIN {X 0,Y 348.057,Z 370.754,A -85,B 0,C 180,E1 -13853.042,E2 -13853.042} C_VEL
LIN {X 0,Y 348.203,Z 370.735,A -85,B 0,C 180,E1 -13857.687,E2 -13857.687} C_VEL
LIN {X 0,Y 348.143,Z 370.743,A -85,B 0,C 180,E1 -13861.157,E2 -13861.157} C_VEL
LIN {X 0,Y 348.195,Z 370.736,A -85,B 0,C 180,E1 -13862.314,E2 -13862.314} C_VEL
LIN {X 0,Y 348.057,Z 370.746,A -85,B 0,C 180,E1 -13866.959,E2 -13866.959} C_VEL
LIN {X 0,Y 347.929,Z 370.765,A -85,B 0,C 180,E1 -13870.475,E2 -13870.475} C_VEL
LIN {X 0,Y 347.901,Z 370.77,A -85,B 0,C 180,E1 -13874.15,E2 -13874.15} C_VEL
LIN {X 0,Y 347.893,Z 370.757,A -85,B 0,C 180,E1 -13878.291,E2 -13878.291} C_VEL
LIN {X 0,Y 347.77,Z 370.784,A -85,B 0,C 180,E1 -13881.627,E2 -13881.627} C_VEL
LIN {X 0,Y 347.746,Z 370.77,A -85,B 0,C 180,E1 -13885.114,E2 -13885.114} C_VEL
LIN {X 0,Y 347.747,Z 370.79,A -85,B 0,C 180,E1 -13887.7,E2 -13887.7} C_VEL
LIN {X 0,Y 347.747,Z 370.776,A -85,B 0,C 180,E1 -13890.349,E2 -13890.349} C_VEL
LIN {X 0,Y 347.751,Z 370.789,A -85,B 0,C 180,E1 -13894.044,E2 -13894.044} C_VEL
LIN {X 0,Y 347.757,Z 370.793,A -85,B 0,C 180,E1 -13897.322,E2 -13897.322} C_VEL
LIN {X 0,Y 347.744,Z 370.79,A -85,B 0,C 180,E1 -13901.601,E2 -13901.601} C_VEL
LIN {X 0,Y 347.752,Z 370.893,A -85,B 0,C 180,E1 -13903.654,E2 -13903.654} C_VEL
LIN {X 0,Y 349.072,Z 375.365,A -85,B 0,C 180,E1 -13905.007,E2 -13905.007} C_VEL
LIN {X 0,Y 356.657,Z 388.411,A -85,B 0,C 180,E1 -13906.309,E2 -13906.309} C_VEL
LIN {X 0,Y 364.717,Z 403.481,A -85,B 0,C 180,E1 -13907.634,E2 -13907.634} C_VEL
LIN {X 0,Y 371.309,Z 417.344,A -85,B 0,C 180,E1 -13908.693,E2 -13908.693} C_VEL
LIN {X 0,Y 367.954,Z 521.831,A -85,B 0,C 180,E1 -13910.751,E2 -13910.751} C_VEL
LIN {X 0,Y 367.283,Z 541.604,A -85,B 0,C 180,E1 -13911.195,E2 -13911.195} C_VEL
LIN {X 0,Y 366.255,Z 556.717,A -85,B 0,C 180,E1 -13911.732,E2 -13911.732} C_VEL
LIN {X 0,Y 364.955,Z 571.397,A -85,B 0,C 180,E1 -13912.482,E2 -13912.482} C_VEL
LIN {X 0,Y 363.348,Z 584.399,A -85,B 0,C 180,E1 -13913.331,E2 -13913.331} C_VEL
LIN {X 0,Y 361.508,Z 598.627,A -85,B 0,C 180,E1 -13914.533,E2 -13914.533} C_VEL
LIN {X 0,Y 359.262,Z 612.203,A -85,B 0,C 180,E1 -13915.946,E2 -13915.946} C_VEL
LIN {X 0,Y 356.959,Z 624.751,A -85,B 0,C 180,E1 -13917.553,E2 -13917.553} C_VEL
LIN {X 0,Y 354.78,Z 636.123,A -85,B 0,C 180,E1 -13919.33,E2 -13919.33} C_VEL
LIN {X 0,Y 352.837,Z 646.109,A -85,B 0,C 180,E1 -13921.215,E2 -13921.215} C_VEL
LIN {X 0,Y 351.012,Z 654.96,A -85,B 0,C 180,E1 -13923.224,E2 -13923.224} C_VEL
LIN {X 0,Y 349.468,Z 662.598,A -85,B 0,C 180,E1 -13925.336,E2 -13925.336} C_VEL
LIN {X 0,Y 348.278,Z 668.845,A -85,B 0,C 180,E1 -13927.455,E2 -13927.455} C_VEL
LIN {X 0,Y 347.296,Z 674.514,A -85,B 0,C 180,E1 -13929.878,E2 -13929.878} C_VEL
LIN {X 0,Y 346.735,Z 678.742,A -85,B 0,C 180,E1 -13932.3,E2 -13932.3} C_VEL
LIN {X 0,Y 346.274,Z 681.661,A -85,B 0,C 180,E1 -13934.701,E2 -13934.701} C_VEL
LIN {X 0,Y 346.179,Z 683.355,A -85,B 0,C 180,E1 -13937.096,E2 -13937.096} C_VEL
LIN {X 0,Y 346.001,Z 683.885,A -85,B 0,C 180,E1 -13939.467,E2 -13939.467} C_VEL
LIN {X 0,Y 346.033,Z 683.228,A -85,B 0,C 180,E1 -13941.827,E2 -13941.827} C_VEL
LIN {X 0,Y 346.253,Z 681.395,A -85,B 0,C 180,E1 -13944.175,E2 -13944.175} C_VEL
LIN {X 0,Y 346.391,Z 678.403,A -85,B 0,C 180,E1 -13946.51,E2 -13946.51} C_VEL
LIN {X 0,Y 346.743,Z 674.184,A -85,B 0,C 180,E1 -13948.839,E2 -13948.839} C_VEL
LIN {X 0,Y 347.282,Z 668.65,A -85,B 0,C 180,E1 -13951.16,E2 -13951.16} C_VEL
LIN {X 0,Y 348.236,Z 661.637,A -85,B 0,C 180,E1 -13953.471,E2 -13953.471} C_VEL
LIN {X 0,Y 349.398,Z 654.141,A -85,B 0,C 180,E1 -13955.483,E2 -13955.483} C_VEL
LIN {X 0,Y 350.742,Z 645.151,A -85,B 0,C 180,E1 -13957.484,E2 -13957.484} C_VEL
LIN {X 0,Y 352.401,Z 634.309,A -85,B 0,C 180,E1 -13959.47,E2 -13959.47} C_VEL
LIN {X 0,Y 354.156,Z 623.173,A -85,B 0,C 180,E1 -13961.156,E2 -13961.156} C_VEL
LIN {X 0,Y 355.798,Z 610.994,A -85,B 0,C 180,E1 -13962.694,E2 -13962.694} C_VEL
LIN {X 0,Y 357.525,Z 597.561,A -85,B 0,C 180,E1 -13964.079,E2 -13964.079} C_VEL
LIN {X 0,Y 358.992,Z 584.397,A -85,B 0,C 180,E1 -13965.18,E2 -13965.18} C_VEL
LIN {X 0,Y 360.377,Z 569.897,A -85,B 0,C 180,E1 -13966.135,E2 -13966.135} C_VEL
LIN {X 0,Y 361.532,Z 554.805,A -85,B 0,C 180,E1 -13966.881,E2 -13966.881} C_VEL
LIN {X 0,Y 362.255,Z 540.102,A -85,B 0,C 180,E1 -13967.391,E2 -13967.391} C_VEL
LIN {X 0,Y 362.535,Z 532.726,A -85,B 0,C 180,E1 -13967.567,E2 -13967.567} C_VEL
LIN {X 0,Y 362.137,Z 526.934,A -85,B 0,C 180,E1 -13967.736,E2 -13967.736} C_VEL
LIN {X 0,Y 357.332,Z 508.275,A -85,B 0,C 180,E1 -13968.491,E2 -13968.491} C_VEL
LIN {X 0,Y 356.831,Z 502.469,A -85,B 0,C 180,E1 -13968.653,E2 -13968.653} C_VEL
LIN {X 0,Y 359.124,Z 414.847,A -85,B 0,C 180,E1 -13970.404,E2 -13970.404} C_VEL
LIN {X 0,Y 350.364,Z 393.8,A -85,B 0,C 180,E1 -13971.626,E2 -13971.626} C_VEL
LIN {X 0,Y 341.461,Z 374.569,A -85,B 0,C 180,E1 -13972.904,E2 -13972.904} C_VEL
LIN {X 0,Y 340.725,Z 371.669,A -85,B 0,C 180,E1 -13973.717,E2 -13973.717} C_VEL
LIN {X 0,Y 340.7,Z 371.672,A -85,B 0,C 180,E1 -13977.499,E2 -13977.499} C_VEL
LIN {X 0,Y 340.699,Z 371.671,A -85,B 0,C 180,E1 -13981.045,E2 -13981.045} C_VEL
LIN {X 0,Y 340.721,Z 371.665,A -85,B 0,C 180,E1 -13985.279,E2 -13985.279} C_VEL
LIN {X 0,Y 340.697,Z 371.67,A -85,B 0,C 180,E1 -13988.382,E2 -13988.382} C_VEL
LIN {X 0,Y 340.697,Z 371.668,A -85,B 0,C 180,E1 -13992.044,E2 -13992.044} C_VEL
LIN {X 0,Y 340.655,Z 371.66,A -85,B 0,C 180,E1 -13996.227,E2 -13996.227} C_VEL
LIN {X 0,Y 340.674,Z 371.672,A -85,B 0,C 180,E1 -13998.688,E2 -13998.688} C_VEL
LIN {X 0,Y 340.721,Z 371.663,A -85,B 0,C 180,E1 -14001.77,E2 -14001.77} C_VEL
LIN {X 0,Y 340.725,Z 371.661,A -85,B 0,C 180,E1 -14005.595,E2 -14005.595} C_VEL
LIN {X 0,Y 340.696,Z 371.673,A -85,B 0,C 180,E1 -14008.954,E2 -14008.954} C_VEL
LIN {X 0,Y 340.713,Z 371.626,A -85,B 0,C 180,E1 -14013.011,E2 -14013.011} C_VEL
LIN {X 0,Y 340.708,Z 371.656,A -85,B 0,C 180,E1 -14016.925,E2 -14016.925} C_VEL
LIN {X 0,Y 340.762,Z 371.659,A -85,B 0,C 180,E1 -14020.731,E2 -14020.731} C_VEL
LIN {X 0,Y 340.82,Z 371.651,A -85,B 0,C 180,E1 -14024.45,E2 -14024.45} C_VEL
LIN {X 0,Y 340.852,Z 371.635,A -85,B 0,C 180,E1 -14028.1,E2 -14028.1} C_VEL
LIN {X 0,Y 340.982,Z 371.636,A -85,B 0,C 180,E1 -14031.704,E2 -14031.704} C_VEL
LIN {X 0,Y 341.015,Z 371.617,A -85,B 0,C 180,E1 -14034.085,E2 -14034.085} C_VEL
LIN {X 0,Y 341.128,Z 371.617,A -85,B 0,C 180,E1 -14037.638,E2 -14037.638} C_VEL
LIN {X 0,Y 341.092,Z 371.609,A -85,B 0,C 180,E1 -14041.18,E2 -14041.18} C_VEL
LIN {X 0,Y 341.159,Z 371.603,A -85,B 0,C 180,E1 -14042.361,E2 -14042.361} C_VEL
LIN {X 0,Y 341.003,Z 371.626,A -85,B 0,C 180,E1 -14047.103,E2 -14047.103} C_VEL
LIN {X 0,Y 340.85,Z 371.649,A -85,B 0,C 180,E1 -14050.694,E2 -14050.694} C_VEL
LIN {X 0,Y 340.819,Z 371.65,A -85,B 0,C 180,E1 -14054.326,E2 -14054.326} C_VEL
LIN {X 0,Y 340.786,Z 371.651,A -85,B 0,C 180,E1 -14058.44,E2 -14058.44} C_VEL
LIN {X 0,Y 340.755,Z 371.655,A -85,B 0,C 180,E1 -14061.856,E2 -14061.856} C_VEL
LIN {X 0,Y 340.72,Z 371.664,A -85,B 0,C 180,E1 -14065.668,E2 -14065.668} C_VEL
LIN {X 0,Y 340.708,Z 371.667,A -85,B 0,C 180,E1 -14069.673,E2 -14069.673} C_VEL
LIN {X 0,Y 340.686,Z 371.669,A -85,B 0,C 180,E1 -14072.435,E2 -14072.435} C_VEL
LIN {X 0,Y 340.717,Z 371.668,A -85,B 0,C 180,E1 -14075.278,E2 -14075.278} C_VEL
LIN {X 0,Y 340.693,Z 371.665,A -85,B 0,C 180,E1 -14078.382,E2 -14078.382} C_VEL
LIN {X 0,Y 340.692,Z 371.671,A -85,B 0,C 180,E1 -14082.044,E2 -14082.044} C_VEL
LIN {X 0,Y 340.65,Z 371.678,A -85,B 0,C 180,E1 -14086.227,E2 -14086.227} C_VEL
LIN {X 0,Y 340.67,Z 371.677,A -85,B 0,C 180,E1 -14088.688,E2 -14088.688} C_VEL
LIN {X 0,Y 340.724,Z 371.707,A -85,B 0,C 180,E1 -14092.52,E2 -14092.52} C_VEL
LIN {X 0,Y 344.204,Z 385.099,A -85,B 0,C 180,E1 -14095.84,E2 -14095.84} C_VEL
LIN {X 0,Y 345.943,Z 392.49,A -85,B 0,C 180,E1 -14097.545,E2 -14097.545} C_VEL
LIN {X 0,Y 353.98,Z 411.777,A -85,B 0,C 180,E1 -14098.694,E2 -14098.694} C_VEL
LIN {X 0,Y 358.707,Z 439.276,A -85,B 0,C 180,E1 -14099.7,E2 -14099.7} C_VEL
LIN {X 0,Y 355.557,Z 559.117,A -85,B 0,C 180,E1 -14102.122,E2 -14102.122} C_VEL
LIN {X 0,Y 354.651,Z 574.476,A -85,B 0,C 180,E1 -14102.645,E2 -14102.645} C_VEL
LIN {X 0,Y 353.357,Z 588.631,A -85,B 0,C 180,E1 -14103.33,E2 -14103.33} C_VEL
LIN {X 0,Y 351.923,Z 602.896,A -85,B 0,C 180,E1 -14104.256,E2 -14104.256} C_VEL
LIN {X 0,Y 350.183,Z 616.706,A -85,B 0,C 180,E1 -14105.39,E2 -14105.39} C_VEL
LIN {X 0,Y 348.446,Z 629.391,A -85,B 0,C 180,E1 -14106.682,E2 -14106.682} C_VEL
LIN {X 0,Y 346.62,Z 641.15,A -85,B 0,C 180,E1 -14108.126,E2 -14108.126} C_VEL
LIN {X 0,Y 345.057,Z 652.091,A -85,B 0,C 180,E1 -14109.742,E2 -14109.742} C_VEL
LIN {X 0,Y 343.526,Z 662.183,A -85,B 0,C 180,E1 -14111.512,E2 -14111.512} C_VEL
LIN {X 0,Y 342.01,Z 672.03,A -85,B 0,C 180,E1 -14113.587,E2 -14113.587} C_VEL
LIN {X 0,Y 340.865,Z 680.338,A -85,B 0,C 180,E1 -14115.707,E2 -14115.707} C_VEL
LIN {X 0,Y 340.008,Z 687.866,A -85,B 0,C 180,E1 -14118.071,E2 -14118.071} C_VEL
LIN {X 0,Y 339.422,Z 693.922,A -85,B 0,C 180,E1 -14120.465,E2 -14120.465} C_VEL
LIN {X 0,Y 339.156,Z 698.574,A -85,B 0,C 180,E1 -14122.858,E2 -14122.858} C_VEL
LIN {X 0,Y 339.044,Z 701.89,A -85,B 0,C 180,E1 -14125.244,E2 -14125.244} C_VEL
LIN {X 0,Y 339.019,Z 703.976,A -85,B 0,C 180,E1 -14127.624,E2 -14127.624} C_VEL
LIN {X 0,Y 339.084,Z 704.898,A -85,B 0,C 180,E1 -14130,E2 -14130} C_VEL
LIN {X 0,Y 339.005,Z 704.677,A -85,B 0,C 180,E1 -14132.376,E2 -14132.376} C_VEL
LIN {X 0,Y 339.025,Z 703.315,A -85,B 0,C 180,E1 -14134.756,E2 -14134.756} C_VEL
LIN {X 0,Y 339.145,Z 700.742,A -85,B 0,C 180,E1 -14137.142,E2 -14137.142} C_VEL
LIN {X 0,Y 339.489,Z 696.97,A -85,B 0,C 180,E1 -14139.533,E2 -14139.533} C_VEL
LIN {X 0,Y 340.165,Z 691.917,A -85,B 0,C 180,E1 -14141.923,E2 -14141.923} C_VEL
LIN {X 0,Y 341.095,Z 685.461,A -85,B 0,C 180,E1 -14144.315,E2 -14144.315} C_VEL
LIN {X 0,Y 342.648,Z 677.426,A -85,B 0,C 180,E1 -14146.688,E2 -14146.688} C_VEL
LIN {X 0,Y 344.31,Z 668.898,A -85,B 0,C 180,E1 -14148.753,E2 -14148.753} C_VEL
LIN {X 0,Y 346.359,Z 659.329,A -85,B 0,C 180,E1 -14150.673,E2 -14150.673} C_VEL
LIN {X 0,Y 348.494,Z 648.244,A -85,B 0,C 180,E1 -14152.53,E2 -14152.53} C_VEL
LIN {X 0,Y 350.745,Z 636.944,A -85,B 0,C 180,E1 -14154.096,E2 -14154.096} C_VEL
LIN {X 0,Y 353.079,Z 624.683,A -85,B 0,C 180,E1 -14155.496,E2 -14155.496} C_VEL
LIN {X 0,Y 355.296,Z 611.32,A -85,B 0,C 180,E1 -14156.744,E2 -14156.744} C_VEL
LIN {X 0,Y 357.29,Z 597.157,A -85,B 0,C 180,E1 -14157.804,E2 -14157.804} C_VEL
LIN {X 0,Y 359.055,Z 582.277,A -85,B 0,C 180,E1 -14158.656,E2 -14158.656} C_VEL
LIN {X 0,Y 360.511,Z 566.846,A -85,B 0,C 180,E1 -14159.287,E2 -14159.287} C_VEL
LIN {X 0,Y 361.386,Z 551.834,A -85,B 0,C 180,E1 -14159.69,E2 -14159.69} C_VEL
LIN {X 0,Y 364.893,Z 440.387,A -85,B 0,C 180,E1 -14161.936,E2 -14161.936} C_VEL
LIN {X 0,Y 361.796,Z 423.426,A -85,B 0,C 180,E1 -14162.691,E2 -14162.691} C_VEL
LIN {X 0,Y 360.892,Z 419.969,A -85,B 0,C 180,E1 -14162.879,E2 -14162.879} C_VEL
LIN {X 0,Y 353.636,Z 404.922,A -85,B 0,C 180,E1 -14164.121,E2 -14164.121} C_VEL
LIN {X 0,Y 346.623,Z 391.427,A -85,B 0,C 180,E1 -14165.395,E2 -14165.395} C_VEL
LIN {X 0,Y 343.407,Z 380.386,A -85,B 0,C 180,E1 -14168.521,E2 -14168.521} C_VEL
LIN {X 0,Y 340.707,Z 371.66,A -85,B 0,C 180,E1 -14171.235,E2 -14171.235} C_VEL
LIN {X 0,Y 340.639,Z 371.677,A -85,B 0,C 180,E1 -14174.546,E2 -14174.546} C_VEL
LIN {X 0,Y 340.692,Z 371.67,A -85,B 0,C 180,E1 -14177.956,E2 -14177.956} C_VEL
LIN {X 0,Y 340.717,Z 371.669,A -85,B 0,C 180,E1 -14181.771,E2 -14181.771} C_VEL
LIN {X 0,Y 340.722,Z 371.663,A -85,B 0,C 180,E1 -14185.596,E2 -14185.596} C_VEL
LIN {X 0,Y 340.695,Z 371.643,A -85,B 0,C 180,E1 -14188.955,E2 -14188.955} C_VEL
LIN {X 0,Y 340.723,Z 371.663,A -85,B 0,C 180,E1 -14193.013,E2 -14193.013} C_VEL
LIN {X 0,Y 340.742,Z 371.665,A -85,B 0,C 180,E1 -14195.638,E2 -14195.638} C_VEL
LIN {X 0,Y 340.741,Z 371.664,A -85,B 0,C 180,E1 -14199.474,E2 -14199.474} C_VEL
LIN {X 0,Y 340.858,Z 371.65,A -85,B 0,C 180,E1 -14201.985,E2 -14201.985} C_VEL
LIN {X 0,Y 340.87,Z 371.648,A -85,B 0,C 180,E1 -14205.706,E2 -14205.706} C_VEL
LIN {X 0,Y 340.849,Z 371.651,A -85,B 0,C 180,E1 -14209.306,E2 -14209.306} C_VEL
LIN {X 0,Y 341.004,Z 371.633,A -85,B 0,C 180,E1 -14212.897,E2 -14212.897} C_VEL
LIN {X 0,Y 340.828,Z 371.646,A -85,B 0,C 180,E1 -14215.269,E2 -14215.269} C_VEL
LIN {X 0,Y 341.165,Z 371.612,A -85,B 0,C 180,E1 -14217.639,E2 -14217.639} C_VEL
LIN {X 0,Y 341.112,Z 371.619,A -85,B 0,C 180,E1 -14221.181,E2 -14221.181} C_VEL
LIN {X 0,Y 341.132,Z 371.615,A -85,B 0,C 180,E1 -14222.362,E2 -14222.362} C_VEL
LIN {X 0,Y 340.993,Z 371.627,A -85,B 0,C 180,E1 -14226.56,E2 -14226.56} C_VEL
LIN {X 0,Y 340.913,Z 371.643,A -85,B 0,C 180,E1 -14229.493,E2 -14229.493} C_VEL
LIN {X 0,Y 340.846,Z 371.652,A -85,B 0,C 180,E1 -14233.11,E2 -14233.11} C_VEL
LIN {X 0,Y 340.789,Z 371.659,A -85,B 0,C 180,E1 -14236.782,E2 -14236.782} C_VEL
LIN {X 0,Y 340.791,Z 371.63,A -85,B 0,C 180,E1 -14239.267,E2 -14239.267} C_VEL
LIN {X 0,Y 340.708,Z 371.669,A -85,B 0,C 180,E1 -14243.075,E2 -14243.075} C_VEL
LIN {X 0,Y 340.727,Z 371.651,A -85,B 0,C 180,E1 -14246.987,E2 -14246.987} C_VEL
LIN {X 0,Y 340.732,Z 371.653,A -85,B 0,C 180,E1 -14249.969,E2 -14249.969} C_VEL
LIN {X 0,Y 340.695,Z 371.672,A -85,B 0,C 180,E1 -14253.847,E2 -14253.847} C_VEL
LIN {X 0,Y 340.703,Z 371.663,A -85,B 0,C 180,E1 -14256.743,E2 -14256.743} C_VEL
LIN {X 0,Y 340.654,Z 371.67,A -85,B 0,C 180,E1 -14260.24,E2 -14260.24} C_VEL
LIN {X 0,Y 340.665,Z 371.67,A -85,B 0,C 180,E1 -14262.787,E2 -14262.787} C_VEL
LIN {X 0,Y 341.87,Z 375.634,A -85,B 0,C 180,E1 -14264.033,E2 -14264.033} C_VEL
LIN {X 0,Y 350.671,Z 390.536,A -85,B 0,C 180,E1 -14265.608,E2 -14265.608} C_VEL
LIN {X 0,Y 359.227,Z 406.476,A -85,B 0,C 180,E1 -14267.066,E2 -14267.066} C_VEL
LIN {X 0,Y 365.368,Z 419.449,A -85,B 0,C 180,E1 -14268.089,E2 -14268.089} C_VEL
LIN {X 0,Y 362.43,Z 511.53,A -85,B 0,C 180,E1 -14269.943,E2 -14269.943} C_VEL
LIN {X 0,Y 361.4,Z 539.769,A -85,B 0,C 180,E1 -14270.531,E2 -14270.531} C_VEL
LIN {X 0,Y 360.377,Z 555.467,A -85,B 0,C 180,E1 -14271.073,E2 -14271.073} C_VEL
LIN {X 0,Y 358.996,Z 570.722,A -85,B 0,C 180,E1 -14271.846,E2 -14271.846} C_VEL
LIN {X 0,Y 357.176,Z 584.737,A -85,B 0,C 180,E1 -14272.767,E2 -14272.767} C_VEL
LIN {X 0,Y 355.269,Z 598.98,A -85,B 0,C 180,E1 -14273.994,E2 -14273.994} C_VEL
LIN {X 0,Y 352.928,Z 612.484,A -85,B 0,C 180,E1 -14275.422,E2 -14275.422} C_VEL
LIN {X 0,Y 350.521,Z 625.02,A -85,B 0,C 180,E1 -14277.053,E2 -14277.053} C_VEL
LIN {X 0,Y 348.385,Z 635.535,A -85,B 0,C 180,E1 -14278.704,E2 -14278.704} C_VEL
LIN {X 0,Y 346.354,Z 645.335,A -85,B 0,C 180,E1 -14280.557,E2 -14280.557} C_VEL
LIN {X 0,Y 344.352,Z 654.585,A -85,B 0,C 180,E1 -14282.664,E2 -14282.664} C_VEL
LIN {X 0,Y 342.729,Z 662.326,A -85,B 0,C 180,E1 -14284.818,E2 -14284.818} C_VEL
LIN {X 0,Y 341.444,Z 668.67,A -85,B 0,C 180,E1 -14286.978,E2 -14286.978} C_VEL
LIN {X 0,Y 340.365,Z 674.429,A -85,B 0,C 180,E1 -14289.45,E2 -14289.45} C_VEL
LIN {X 0,Y 339.694,Z 679.036,A -85,B 0,C 180,E1 -14292.122,E2 -14292.122} C_VEL
LIN {X 0,Y 339.226,Z 681.745,A -85,B 0,C 180,E1 -14294.376,E2 -14294.376} C_VEL
LIN {X 0,Y 339.087,Z 683.566,A -85,B 0,C 180,E1 -14296.944,E2 -14296.944} C_VEL
LIN {X 0,Y 338.933,Z 684.114,A -85,B 0,C 180,E1 -14299.244,E2 -14299.244} C_VEL
LIN {X 0,Y 338.934,Z 683.507,A -85,B 0,C 180,E1 -14301.654,E2 -14301.654} C_VEL
LIN {X 0,Y 339.174,Z 681.749,A -85,B 0,C 180,E1 -14304.053,E2 -14304.053} C_VEL
LIN {X 0,Y 339.299,Z 678.837,A -85,B 0,C 180,E1 -14306.437,E2 -14306.437} C_VEL
LIN {X 0,Y 339.662,Z 674.7,A -85,B 0,C 180,E1 -14308.814,E2 -14308.814} C_VEL
LIN {X 0,Y 340.207,Z 669.255,A -85,B 0,C 180,E1 -14311.184,E2 -14311.184} C_VEL
LIN {X 0,Y 341.173,Z 662.339,A -85,B 0,C 180,E1 -14313.543,E2 -14313.543} C_VEL
LIN {X 0,Y 342.374,Z 654.939,A -85,B 0,C 180,E1 -14315.596,E2 -14315.596} C_VEL
LIN {X 0,Y 343.749,Z 646.035,A -85,B 0,C 180,E1 -14317.637,E2 -14317.637} C_VEL
LIN {X 0,Y 345.454,Z 635.349,A -85,B 0,C 180,E1 -14319.662,E2 -14319.662} C_VEL
LIN {X 0,Y 347.413,Z 623.336,A -85,B 0,C 180,E1 -14321.523,E2 -14321.523} C_VEL
LIN {X 0,Y 349.119,Z 611.141,A -85,B 0,C 180,E1 -14323.089,E2 -14323.089} C_VEL
LIN {X 0,Y 350.926,Z 597.686,A -85,B 0,C 180,E1 -14324.498,E2 -14324.498} C_VEL
LIN {X 0,Y 352.446,Z 584.507,A -85,B 0,C 180,E1 -14325.617,E2 -14325.617} C_VEL
LIN {X 0,Y 353.872,Z 569.98,A -85,B 0,C 180,E1 -14326.588,E2 -14326.588} C_VEL
LIN {X 0,Y 355.074,Z 554.835,A -85,B 0,C 180,E1 -14327.346,E2 -14327.346} C_VEL
LIN {X 0,Y 355.813,Z 540.06,A -85,B 0,C 180,E1 -14327.865,E2 -14327.865} C_VEL
LIN {X 0,Y 356.831,Z 502.469,A -85,B 0,C 180,E1 -14328.653,E2 -14328.653} C_VEL
LIN {X 0,Y 356.366,Z 496.668,A -85,B 0,C 180,E1 -14328.817,E2 -14328.817} C_VEL
LIN {X 0,Y 351.806,Z 477.984,A -85,B 0,C 180,E1 -14329.594,E2 -14329.594} C_VEL
LIN {X 0,Y 351.353,Z 472.183,A -85,B 0,C 180,E1 -14329.761,E2 -14329.761} C_VEL
LIN {X 0,Y 352.784,Z 416.596,A -85,B 0,C 180,E1 -14330.896,E2 -14330.896} C_VEL
LIN {X 0,Y 343.436,Z 394.251,A -85,B 0,C 180,E1 -14332.241,E2 -14332.241} C_VEL
LIN {X 0,Y 335.258,Z 377.125,A -85,B 0,C 180,E1 -14333.433,E2 -14333.433} C_VEL
LIN {X 0,Y 334.183,Z 374.698,A -85,B 0,C 180,E1 -14333.634,E2 -14333.634} C_VEL
LIN {X 0,Y 333.695,Z 372.544,A -85,B 0,C 180,E1 -14334.249,E2 -14334.249} C_VEL
LIN {X 0,Y 333.655,Z 372.549,A -85,B 0,C 180,E1 -14337.787,E2 -14337.787} C_VEL
LIN {X 0,Y 333.662,Z 372.545,A -85,B 0,C 180,E1 -14340.366,E2 -14340.366} C_VEL
LIN {X 0,Y 333.641,Z 372.542,A -85,B 0,C 180,E1 -14343.208,E2 -14343.208} C_VEL
LIN {X 0,Y 333.679,Z 372.535,A -85,B 0,C 180,E1 -14346.139,E2 -14346.139} C_VEL
LIN {X 0,Y 333.623,Z 372.55,A -85,B 0,C 180,E1 -14349.196,E2 -14349.196} C_VEL
LIN {X 0,Y 333.632,Z 372.549,A -85,B 0,C 180,E1 -14352.499,E2 -14352.499} C_VEL
LIN {X 0,Y 333.599,Z 372.538,A -85,B 0,C 180,E1 -14355.954,E2 -14355.954} C_VEL
LIN {X 0,Y 333.606,Z 372.556,A -85,B 0,C 180,E1 -14359.324,E2 -14359.324} C_VEL
LIN {X 0,Y 333.665,Z 372.547,A -85,B 0,C 180,E1 -14363.168,E2 -14363.168} C_VEL
LIN {X 0,Y 333.676,Z 372.541,A -85,B 0,C 180,E1 -14365.341,E2 -14365.341} C_VEL
LIN {X 0,Y 333.632,Z 372.553,A -85,B 0,C 180,E1 -14368.221,E2 -14368.221} C_VEL
LIN {X 0,Y 333.654,Z 372.533,A -85,B 0,C 180,E1 -14371.022,E2 -14371.022} C_VEL
LIN {X 0,Y 333.665,Z 372.509,A -85,B 0,C 180,E1 -14375.085,E2 -14375.085} C_VEL
LIN {X 0,Y 333.674,Z 372.545,A -85,B 0,C 180,E1 -14379.018,E2 -14379.018} C_VEL
LIN {X 0,Y 333.744,Z 372.526,A -85,B 0,C 180,E1 -14381.586,E2 -14381.586} C_VEL
LIN {X 0,Y 333.811,Z 372.53,A -85,B 0,C 180,E1 -14385.576,E2 -14385.576} C_VEL
LIN {X 0,Y 333.82,Z 372.51,A -85,B 0,C 180,E1 -14389.077,E2 -14389.077} C_VEL
LIN {X 0,Y 333.958,Z 372.506,A -85,B 0,C 180,E1 -14392.745,E2 -14392.745} C_VEL
LIN {X 0,Y 333.781,Z 372.516,A -85,B 0,C 180,E1 -14395.168,E2 -14395.168} C_VEL
LIN {X 0,Y 334.068,Z 372.495,A -85,B 0,C 180,E1 -14397.588,E2 -14397.588} C_VEL
LIN {X 0,Y 334.063,Z 372.484,A -85,B 0,C 180,E1 -14401.205,E2 -14401.205} C_VEL
LIN {X 0,Y 334.095,Z 372.483,A -85,B 0,C 180,E1 -14402.411,E2 -14402.411} C_VEL
LIN {X 0,Y 333.991,Z 372.502,A -85,B 0,C 180,E1 -14406.039,E2 -14406.039} C_VEL
LIN {X 0,Y 333.822,Z 372.526,A -85,B 0,C 180,E1 -14409.696,E2 -14409.696} C_VEL
LIN {X 0,Y 333.788,Z 372.52,A -85,B 0,C 180,E1 -14413.391,E2 -14413.391} C_VEL
LIN {X 0,Y 333.702,Z 372.536,A -85,B 0,C 180,E1 -14417.148,E2 -14417.148} C_VEL
LIN {X 0,Y 333.721,Z 372.538,A -85,B 0,C 180,E1 -14419.691,E2 -14419.691} C_VEL
LIN {X 0,Y 333.691,Z 372.534,A -85,B 0,C 180,E1 -14422.278,E2 -14422.278} C_VEL
LIN {X 0,Y 333.69,Z 372.542,A -85,B 0,C 180,E1 -14425.089,E2 -14425.089} C_VEL
LIN {X 0,Y 333.654,Z 372.547,A -85,B 0,C 180,E1 -14428.977,E2 -14428.977} C_VEL
LIN {X 0,Y 333.644,Z 372.546,A -85,B 0,C 180,E1 -14432.586,E2 -14432.586} C_VEL
LIN {X 0,Y 333.674,Z 372.544,A -85,B 0,C 180,E1 -14436.139,E2 -14436.139} C_VEL
LIN {X 0,Y 333.601,Z 372.543,A -85,B 0,C 180,E1 -14439.198,E2 -14439.198} C_VEL
LIN {X 0,Y 333.628,Z 372.549,A -85,B 0,C 180,E1 -14442.499,E2 -14442.499} C_VEL
LIN {X 0,Y 333.594,Z 372.557,A -85,B 0,C 180,E1 -14445.954,E2 -14445.954} C_VEL
LIN {X 0,Y 333.601,Z 372.553,A -85,B 0,C 180,E1 -14449.324,E2 -14449.324} C_VEL
LIN {X 0,Y 333.694,Z 372.624,A -85,B 0,C 180,E1 -14451.972,E2 -14451.972} C_VEL
LIN {X 0,Y 337.252,Z 386.248,A -85,B 0,C 180,E1 -14455.447,E2 -14455.447} C_VEL
LIN {X 0,Y 338.608,Z 392.103,A -85,B 0,C 180,E1 -14456.852,E2 -14456.852} C_VEL
LIN {X 0,Y 347.932,Z 414.23,A -85,B 0,C 180,E1 -14458.227,E2 -14458.227} C_VEL
LIN {X 0,Y 352.36,Z 439.932,A -85,B 0,C 180,E1 -14459.193,E2 -14459.193} C_VEL
LIN {X 0,Y 349.117,Z 559.106,A -85,B 0,C 180,E1 -14461.643,E2 -14461.643} C_VEL
LIN {X 0,Y 348.173,Z 574.394,A -85,B 0,C 180,E1 -14462.174,E2 -14462.174} C_VEL
LIN {X 0,Y 346.725,Z 589.621,A -85,B 0,C 180,E1 -14462.931,E2 -14462.931} C_VEL
LIN {X 0,Y 345.246,Z 603.76,A -85,B 0,C 180,E1 -14463.883,E2 -14463.883} C_VEL
LIN {X 0,Y 343.452,Z 617.353,A -85,B 0,C 180,E1 -14465.036,E2 -14465.036} C_VEL
LIN {X 0,Y 341.44,Z 631.176,A -85,B 0,C 180,E1 -14466.496,E2 -14466.496} C_VEL
LIN {X 0,Y 339.447,Z 643.68,A -85,B 0,C 180,E1 -14468.119,E2 -14468.119} C_VEL
LIN {X 0,Y 337.717,Z 655.072,A -85,B 0,C 180,E1 -14469.918,E2 -14469.918} C_VEL
LIN {X 0,Y 335.924,Z 666.108,A -85,B 0,C 180,E1 -14472.026,E2 -14472.026} C_VEL
LIN {X 0,Y 334.586,Z 675.272,A -85,B 0,C 180,E1 -14474.153,E2 -14474.153} C_VEL
LIN {X 0,Y 333.416,Z 683.837,A -85,B 0,C 180,E1 -14476.593,E2 -14476.593} C_VEL
LIN {X 0,Y 332.585,Z 690.699,A -85,B 0,C 180,E1 -14479.036,E2 -14479.036} C_VEL
LIN {X 0,Y 332.222,Z 696.08,A -85,B 0,C 180,E1 -14481.484,E2 -14481.484} C_VEL
LIN {X 0,Y 332.03,Z 700.079,A -85,B 0,C 180,E1 -14483.925,E2 -14483.925} C_VEL
LIN {X 0,Y 331.98,Z 702.804,A -85,B 0,C 180,E1 -14486.359,E2 -14486.359} C_VEL
LIN {X 0,Y 331.947,Z 704.335,A -85,B 0,C 180,E1 -14488.787,E2 -14488.787} C_VEL
LIN {X 0,Y 331.94,Z 704.718,A -85,B 0,C 180,E1 -14491.213,E2 -14491.213} C_VEL
LIN {X 0,Y 331.949,Z 703.965,A -85,B 0,C 180,E1 -14493.642,E2 -14493.642} C_VEL
LIN {X 0,Y 331.992,Z 702.017,A -85,B 0,C 180,E1 -14496.076,E2 -14496.076} C_VEL
LIN {X 0,Y 332.24,Z 698.888,A -85,B 0,C 180,E1 -14498.515,E2 -14498.515} C_VEL
LIN {X 0,Y 332.693,Z 694.529,A -85,B 0,C 180,E1 -14500.96,E2 -14500.96} C_VEL
LIN {X 0,Y 333.614,Z 688.836,A -85,B 0,C 180,E1 -14503.399,E2 -14503.399} C_VEL
LIN {X 0,Y 334.934,Z 681.663,A -85,B 0,C 180,E1 -14505.83,E2 -14505.83} C_VEL
LIN {X 0,Y 336.523,Z 674.026,A -85,B 0,C 180,E1 -14507.941,E2 -14507.941} C_VEL
LIN {X 0,Y 338.555,Z 664.876,A -85,B 0,C 180,E1 -14510.031,E2 -14510.031} C_VEL
LIN {X 0,Y 340.834,Z 653.861,A -85,B 0,C 180,E1 -14512.106,E2 -14512.106} C_VEL
LIN {X 0,Y 343.221,Z 642.58,A -85,B 0,C 180,E1 -14513.854,E2 -14513.854} C_VEL
LIN {X 0,Y 345.425,Z 631.443,A -85,B 0,C 180,E1 -14515.294,E2 -14515.294} C_VEL
LIN {X 0,Y 347.994,Z 618.075,A -85,B 0,C 180,E1 -14516.702,E2 -14516.702} C_VEL
LIN {X 0,Y 350.126,Z 604.651,A -85,B 0,C 180,E1 -14517.851,E2 -14517.851} C_VEL
LIN {X 0,Y 352.025,Z 590.733,A -85,B 0,C 180,E1 -14518.793,E2 -14518.793} C_VEL
LIN {X 0,Y 353.619,Z 576.817,A -85,B 0,C 180,E1 -14519.506,E2 -14519.506} C_VEL
LIN {X 0,Y 354.834,Z 562.158,A -85,B 0,C 180,E1 -14520.048,E2 -14520.048} C_VEL
LIN {X 0,Y 355.721,Z 542.886,A -85,B 0,C 180,E1 -14520.498,E2 -14520.498} C_VEL
LIN {X 0,Y 359.039,Z 440.969,A -85,B 0,C 180,E1 -14522.583,E2 -14522.583} C_VEL
LIN {X 0,Y 355.842,Z 423.897,A -85,B 0,C 180,E1 -14523.377,E2 -14523.377} C_VEL
LIN {X 0,Y 349.301,Z 410.122,A -85,B 0,C 180,E1 -14524.535,E2 -14524.535} C_VEL
LIN {X 0,Y 341.529,Z 395.354,A -85,B 0,C 180,E1 -14525.953,E2 -14525.953} C_VEL
LIN {X 0,Y 339.269,Z 391.205,A -85,B 0,C 180,E1 -14526.391,E2 -14526.391} C_VEL
LIN {X 0,Y 336.968,Z 383.186,A -85,B 0,C 180,E1 -14528.733,E2 -14528.733} C_VEL
LIN {X 0,Y 333.659,Z 372.535,A -85,B 0,C 180,E1 -14532.105,E2 -14532.105} C_VEL
LIN {X 0,Y 333.594,Z 372.555,A -85,B 0,C 180,E1 -14535.955,E2 -14535.955} C_VEL
LIN {X 0,Y 333.601,Z 372.556,A -85,B 0,C 180,E1 -14539.325,E2 -14539.325} C_VEL
LIN {X 0,Y 333.661,Z 372.527,A -85,B 0,C 180,E1 -14543.169,E2 -14543.169} C_VEL
LIN {X 0,Y 333.639,Z 372.547,A -85,B 0,C 180,E1 -14546.792,E2 -14546.792} C_VEL
LIN {X 0,Y 333.661,Z 372.52,A -85,B 0,C 180,E1 -14549.723,E2 -14549.723} C_VEL
LIN {X 0,Y 333.66,Z 372.54,A -85,B 0,C 180,E1 -14553.748,E2 -14553.748} C_VEL
LIN {X 0,Y 333.663,Z 372.543,A -85,B 0,C 180,E1 -14556.41,E2 -14556.41} C_VEL
LIN {X 0,Y 333.733,Z 372.533,A -85,B 0,C 180,E1 -14560.31,E2 -14560.31} C_VEL
LIN {X 0,Y 333.747,Z 372.535,A -85,B 0,C 180,E1 -14562.854,E2 -14562.854} C_VEL
LIN {X 0,Y 333.797,Z 372.528,A -85,B 0,C 180,E1 -14566.609,E2 -14566.609} C_VEL
LIN {X 0,Y 333.822,Z 372.527,A -85,B 0,C 180,E1 -14570.304,E2 -14570.304} C_VEL
LIN {X 0,Y 333.992,Z 372.507,A -85,B 0,C 180,E1 -14573.961,E2 -14573.961} C_VEL
LIN {X 0,Y 334.102,Z 372.492,A -85,B 0,C 180,E1 -14577.589,E2 -14577.589} C_VEL
LIN {X 0,Y 334.08,Z 372.495,A -85,B 0,C 180,E1 -14581.206,E2 -14581.206} C_VEL
LIN {X 0,Y 333.815,Z 372.518,A -85,B 0,C 180,E1 -14583.622,E2 -14583.622} C_VEL
LIN {X 0,Y 333.96,Z 372.505,A -85,B 0,C 180,E1 -14586.553,E2 -14586.553} C_VEL
LIN {X 0,Y 333.85,Z 372.524,A -85,B 0,C 180,E1 -14589.696,E2 -14589.696} C_VEL
LIN {X 0,Y 333.799,Z 372.529,A -85,B 0,C 180,E1 -14593.392,E2 -14593.392} C_VEL
LIN {X 0,Y 333.749,Z 372.534,A -85,B 0,C 180,E1 -14597.147,E2 -14597.147} C_VEL
LIN {X 0,Y 333.734,Z 372.507,A -85,B 0,C 180,E1 -14599.691,E2 -14599.691} C_VEL
LIN {X 0,Y 333.648,Z 372.548,A -85,B 0,C 180,E1 -14603.593,E2 -14603.593} C_VEL
LIN {X 0,Y 333.677,Z 372.541,A -85,B 0,C 180,E1 -14607.605,E2 -14607.605} C_VEL
LIN {X 0,Y 333.662,Z 372.529,A -85,B 0,C 180,E1 -14610.366,E2 -14610.366} C_VEL
LIN {X 0,Y 333.64,Z 372.552,A -85,B 0,C 180,E1 -14613.209,E2 -14613.209} C_VEL
LIN {X 0,Y 333.676,Z 372.531,A -85,B 0,C 180,E1 -14616.14,E2 -14616.14} C_VEL
LIN {X 0,Y 333.604,Z 372.542,A -85,B 0,C 180,E1 -14619.199,E2 -14619.199} C_VEL
LIN {X 0,Y 333.697,Z 372.738,A -85,B 0,C 180,E1 -14621.967,E2 -14621.967} C_VEL
LIN {X 0,Y 334.624,Z 375.893,A -85,B 0,C 180,E1 -14622.994,E2 -14622.994} C_VEL
LIN {X 0,Y 344.943,Z 393.017,A -85,B 0,C 180,E1 -14624.919,E2 -14624.919} C_VEL
LIN {X 0,Y 354.201,Z 410.335,A -85,B 0,C 180,E1 -14626.555,E2 -14626.555} C_VEL
LIN {X 0,Y 359.613,Z 421.847,A -85,B 0,C 180,E1 -14627.488,E2 -14627.488} C_VEL
LIN {X 0,Y 355.979,Z 525.253,A -85,B 0,C 180,E1 -14629.577,E2 -14629.577} C_VEL
LIN {X 0,Y 355.293,Z 543.971,A -85,B 0,C 180,E1 -14630.039,E2 -14630.039} C_VEL
LIN {X 0,Y 354.128,Z 558.925,A -85,B 0,C 180,E1 -14630.611,E2 -14630.611} C_VEL
LIN {X 0,Y 352.615,Z 573.821,A -85,B 0,C 180,E1 -14631.422,E2 -14631.422} C_VEL
LIN {X 0,Y 350.815,Z 586.938,A -85,B 0,C 180,E1 -14632.337,E2 -14632.337} C_VEL
LIN {X 0,Y 349,Z 599.748,A -85,B 0,C 180,E1 -14633.475,E2 -14633.475} C_VEL
LIN {X 0,Y 346.623,Z 612.792,A -85,B 0,C 180,E1 -14634.878,E2 -14634.878} C_VEL
LIN {X 0,Y 344.334,Z 624.29,A -85,B 0,C 180,E1 -14636.383,E2 -14636.383} C_VEL
LIN {X 0,Y 342.064,Z 634.9,A -85,B 0,C 180,E1 -14638.058,E2 -14638.058} C_VEL
LIN {X 0,Y 339.964,Z 644.677,A -85,B 0,C 180,E1 -14639.913,E2 -14639.913} C_VEL
LIN {X 0,Y 337.763,Z 654.203,A -85,B 0,C 180,E1 -14642.085,E2 -14642.085} C_VEL
LIN {X 0,Y 336.112,Z 661.658,A -85,B 0,C 180,E1 -14644.158,E2 -14644.158} C_VEL
LIN {X 0,Y 334.655,Z 668.5,A -85,B 0,C 180,E1 -14646.483,E2 -14646.483} C_VEL
LIN {X 0,Y 333.465,Z 674.351,A -85,B 0,C 180,E1 -14649.005,E2 -14649.005} C_VEL
LIN {X 0,Y 332.713,Z 678.75,A -85,B 0,C 180,E1 -14651.527,E2 -14651.527} C_VEL
LIN {X 0,Y 332.187,Z 681.831,A -85,B 0,C 180,E1 -14654.036,E2 -14654.036} C_VEL
LIN {X 0,Y 331.998,Z 683.683,A -85,B 0,C 180,E1 -14656.535,E2 -14656.535} C_VEL
LIN {X 0,Y 331.843,Z 684.319,A -85,B 0,C 180,E1 -14659.012,E2 -14659.012} C_VEL
LIN {X 0,Y 331.819,Z 683.785,A -85,B 0,C 180,E1 -14661.474,E2 -14661.474} C_VEL
LIN {X 0,Y 332.09,Z 681.958,A -85,B 0,C 180,E1 -14664.083,E2 -14664.083} C_VEL
LIN {X 0,Y 332.21,Z 679.269,A -85,B 0,C 180,E1 -14666.361,E2 -14666.361} C_VEL
LIN {X 0,Y 332.584,Z 675.213,A -85,B 0,C 180,E1 -14668.789,E2 -14668.789} C_VEL
LIN {X 0,Y 333.134,Z 669.853,A -85,B 0,C 180,E1 -14671.209,E2 -14671.209} C_VEL
LIN {X 0,Y 334.111,Z 663.03,A -85,B 0,C 180,E1 -14673.618,E2 -14673.618} C_VEL
LIN {X 0,Y 335.501,Z 654.526,A -85,B 0,C 180,E1 -14676.012,E2 -14676.012} C_VEL
LIN {X 0,Y 336.985,Z 645.518,A -85,B 0,C 180,E1 -14678.093,E2 -14678.093} C_VEL
LIN {X 0,Y 338.787,Z 634.655,A -85,B 0,C 180,E1 -14680.156,E2 -14680.156} C_VEL
LIN {X 0,Y 340.671,Z 623.496,A -85,B 0,C 180,E1 -14681.906,E2 -14681.906} C_VEL
LIN {X 0,Y 342.432,Z 611.292,A -85,B 0,C 180,E1 -14683.501,E2 -14683.501} C_VEL
LIN {X 0,Y 344.34,Z 597.811,A -85,B 0,C 180,E1 -14684.932,E2 -14684.932} C_VEL
LIN {X 0,Y 345.917,Z 584.617,A -85,B 0,C 180,E1 -14686.071,E2 -14686.071} C_VEL
LIN {X 0,Y 347.389,Z 570.061,A -85,B 0,C 180,E1 -14687.059,E2 -14687.059} C_VEL
LIN {X 0,Y 348.632,Z 554.863,A -85,B 0,C 180,E1 -14687.828,E2 -14687.828} C_VEL
LIN {X 0,Y 349.393,Z 540.016,A -85,B 0,C 180,E1 -14688.356,E2 -14688.356} C_VEL
LIN {X 0,Y 351.353,Z 472.183,A -85,B 0,C 180,E1 -14689.761,E2 -14689.761} C_VEL
LIN {X 0,Y 350.906,Z 466.383,A -85,B 0,C 180,E1 -14689.928,E2 -14689.928} C_VEL
LIN {X 0,Y 346.376,Z 447.713,A -85,B 0,C 180,E1 -14690.735,E2 -14690.735} C_VEL
LIN {X 0,Y 345.868,Z 441.916,A -85,B 0,C 180,E1 -14690.912,E2 -14690.912} C_VEL
LIN {X 0,Y 346.447,Z 418.286,A -85,B 0,C 180,E1 -14691.408,E2 -14691.408} C_VEL
LIN {X 0,Y 337.529,Z 397.073,A -85,B 0,C 180,E1 -14692.729,E2 -14692.729} C_VEL
LIN {X 0,Y 329.772,Z 380.812,A -85,B 0,C 180,E1 -14693.894,E2 -14693.894} C_VEL
LIN {X 0,Y 327.023,Z 374.96,A -85,B 0,C 180,E1 -14694.354,E2 -14694.354} C_VEL
LIN {X 0,Y 326.624,Z 373.422,A -85,B 0,C 180,E1 -14694.809,E2 -14694.809} C_VEL
LIN {X 0,Y 326.603,Z 373.427,A -85,B 0,C 180,E1 -14698.256,E2 -14698.256} C_VEL
LIN {X 0,Y 326.578,Z 373.43,A -85,B 0,C 180,E1 -14701.097,E2 -14701.097} C_VEL
LIN {X 0,Y 326.611,Z 373.427,A -85,B 0,C 180,E1 -14704.019,E2 -14704.019} C_VEL
LIN {X 0,Y 326.626,Z 373.417,A -85,B 0,C 180,E1 -14707.237,E2 -14707.237} C_VEL
LIN {X 0,Y 326.547,Z 373.42,A -85,B 0,C 180,E1 -14711.124,E2 -14711.124} C_VEL
LIN {X 0,Y 326.564,Z 373.433,A -85,B 0,C 180,E1 -14713.525,E2 -14713.525} C_VEL
LIN {X 0,Y 326.577,Z 373.417,A -85,B 0,C 180,E1 -14717.028,E2 -14717.028} C_VEL
LIN {X 0,Y 326.574,Z 373.424,A -85,B 0,C 180,E1 -14720.781,E2 -14720.781} C_VEL
LIN {X 0,Y 326.613,Z 373.423,A -85,B 0,C 180,E1 -14724.48,E2 -14724.48} C_VEL
LIN {X 0,Y 326.611,Z 373.425,A -85,B 0,C 180,E1 -14727.455,E2 -14727.455} C_VEL
LIN {X 0,Y 326.618,Z 373.417,A -85,B 0,C 180,E1 -14730.336,E2 -14730.336} C_VEL
LIN {X 0,Y 326.602,Z 373.38,A -85,B 0,C 180,E1 -14734.508,E2 -14734.508} C_VEL
LIN {X 0,Y 326.621,Z 373.422,A -85,B 0,C 180,E1 -14738.543,E2 -14738.543} C_VEL
LIN {X 0,Y 326.71,Z 373.407,A -85,B 0,C 180,E1 -14741.175,E2 -14741.175} C_VEL
LIN {X 0,Y 326.766,Z 373.407,A -85,B 0,C 180,E1 -14745.433,E2 -14745.433} C_VEL
LIN {X 0,Y 326.761,Z 373.388,A -85,B 0,C 180,E1 -14748.838,E2 -14748.838} C_VEL
LIN {X 0,Y 326.915,Z 373.383,A -85,B 0,C 180,E1 -14752.588,E2 -14752.588} C_VEL
LIN {X 0,Y 326.749,Z 373.391,A -85,B 0,C 180,E1 -14755.064,E2 -14755.064} C_VEL
LIN {X 0,Y 327.012,Z 373.374,A -85,B 0,C 180,E1 -14757.536,E2 -14757.536} C_VEL
LIN {X 0,Y 327.033,Z 373.359,A -85,B 0,C 180,E1 -14761.231,E2 -14761.231} C_VEL
LIN {X 0,Y 327.036,Z 373.362,A -85,B 0,C 180,E1 -14762.463,E2 -14762.463} C_VEL
LIN {X 0,Y 326.945,Z 373.379,A -85,B 0,C 180,E1 -14766.17,E2 -14766.17} C_VEL
LIN {X 0,Y 326.785,Z 373.404,A -85,B 0,C 180,E1 -14769.907,E2 -14769.907} C_VEL
LIN {X 0,Y 326.744,Z 373.399,A -85,B 0,C 180,E1 -14773.686,E2 -14773.686} C_VEL
LIN {X 0,Y 326.652,Z 373.411,A -85,B 0,C 180,E1 -14777.53,E2 -14777.53} C_VEL
LIN {X 0,Y 326.655,Z 373.417,A -85,B 0,C 180,E1 -14780.135,E2 -14780.135} C_VEL
LIN {X 0,Y 326.617,Z 373.415,A -85,B 0,C 180,E1 -14782.787,E2 -14782.787} C_VEL
LIN {X 0,Y 326.635,Z 373.419,A -85,B 0,C 180,E1 -14785.488,E2 -14785.488} C_VEL
LIN {X 0,Y 326.617,Z 373.422,A -85,B 0,C 180,E1 -14789.663,E2 -14789.663} C_VEL
LIN {X 0,Y 326.617,Z 373.421,A -85,B 0,C 180,E1 -14792.945,E2 -14792.945} C_VEL
LIN {X 0,Y 326.611,Z 373.424,A -85,B 0,C 180,E1 -14795.519,E2 -14795.519} C_VEL
LIN {X 0,Y 326.57,Z 373.418,A -85,B 0,C 180,E1 -14799.218,E2 -14799.218} C_VEL
LIN {X 0,Y 326.572,Z 373.428,A -85,B 0,C 180,E1 -14802.971,E2 -14802.971} C_VEL
LIN {X 0,Y 326.572,Z 373.433,A -85,B 0,C 180,E1 -14807.028,E2 -14807.028} C_VEL
LIN {X 0,Y 326.617,Z 373.499,A -85,B 0,C 180,E1 -14811.39,E2 -14811.39} C_VEL
LIN {X 0,Y 330.226,Z 386.966,A -85,B 0,C 180,E1 -14814.926,E2 -14814.926} C_VEL
LIN {X 0,Y 331.338,Z 391.875,A -85,B 0,C 180,E1 -14816.135,E2 -14816.135} C_VEL
LIN {X 0,Y 340.617,Z 413.526,A -85,B 0,C 180,E1 -14817.551,E2 -14817.551} C_VEL
LIN {X 0,Y 342.097,Z 417.475,A -85,B 0,C 180,E1 -14817.779,E2 -14817.779} C_VEL
LIN {X 0,Y 346.016,Z 440.529,A -85,B 0,C 180,E1 -14818.666,E2 -14818.666} C_VEL
LIN {X 0,Y 342.701,Z 559.005,A -85,B 0,C 180,E1 -14821.146,E2 -14821.146} C_VEL
LIN {X 0,Y 341.722,Z 574.261,A -85,B 0,C 180,E1 -14821.685,E2 -14821.685} C_VEL
LIN {X 0,Y 340.325,Z 588.472,A -85,B 0,C 180,E1 -14822.396,E2 -14822.396} C_VEL
LIN {X 0,Y 338.886,Z 601.783,A -85,B 0,C 180,E1 -14823.287,E2 -14823.287} C_VEL
LIN {X 0,Y 337.162,Z 614.786,A -85,B 0,C 180,E1 -14824.372,E2 -14824.372} C_VEL
LIN {X 0,Y 335.31,Z 627.752,A -85,B 0,C 180,E1 -14825.711,E2 -14825.711} C_VEL
LIN {X 0,Y 333.299,Z 639.714,A -85,B 0,C 180,E1 -14827.203,E2 -14827.203} C_VEL
LIN {X 0,Y 331.527,Z 650.815,A -85,B 0,C 180,E1 -14828.876,E2 -14828.876} C_VEL
LIN {X 0,Y 329.901,Z 661.051,A -85,B 0,C 180,E1 -14830.719,E2 -14830.719} C_VEL
LIN {X 0,Y 328.232,Z 671.02,A -85,B 0,C 180,E1 -14832.878,E2 -14832.878} C_VEL
LIN {X 0,Y 326.983,Z 679.325,A -85,B 0,C 180,E1 -14835.053,E2 -14835.053} C_VEL
LIN {X 0,Y 326,Z 687.061,A -85,B 0,C 180,E1 -14837.55,E2 -14837.55} C_VEL
LIN {X 0,Y 325.319,Z 693.199,A -85,B 0,C 180,E1 -14840.048,E2 -14840.048} C_VEL
LIN {X 0,Y 324.996,Z 697.905,A -85,B 0,C 180,E1 -14842.545,E2 -14842.545} C_VEL
LIN {X 0,Y 324.864,Z 701.291,A -85,B 0,C 180,E1 -14845.036,E2 -14845.036} C_VEL
LIN {X 0,Y 324.852,Z 703.451,A -85,B 0,C 180,E1 -14847.52,E2 -14847.52} C_VEL
LIN {X 0,Y 324.891,Z 704.442,A -85,B 0,C 180,E1 -14850,E2 -14850} C_VEL
LIN {X 0,Y 324.838,Z 704.291,A -85,B 0,C 180,E1 -14852.48,E2 -14852.48} C_VEL
LIN {X 0,Y 324.848,Z 702.969,A -85,B 0,C 180,E1 -14854.964,E2 -14854.964} C_VEL
LIN {X 0,Y 324.977,Z 700.462,A -85,B 0,C 180,E1 -14857.456,E2 -14857.456} C_VEL
LIN {X 0,Y 325.389,Z 696.768,A -85,B 0,C 180,E1 -14859.95,E2 -14859.95} C_VEL
LIN {X 0,Y 326.17,Z 691.799,A -85,B 0,C 180,E1 -14862.443,E2 -14862.443} C_VEL
LIN {X 0,Y 327.231,Z 685.43,A -85,B 0,C 180,E1 -14864.935,E2 -14864.935} C_VEL
LIN {X 0,Y 328.974,Z 677.494,A -85,B 0,C 180,E1 -14867.403,E2 -14867.403} C_VEL
LIN {X 0,Y 330.833,Z 669.081,A -85,B 0,C 180,E1 -14869.547,E2 -14869.547} C_VEL
LIN {X 0,Y 332.872,Z 660.427,A -85,B 0,C 180,E1 -14871.389,E2 -14871.389} C_VEL
LIN {X 0,Y 335.4,Z 648.718,A -85,B 0,C 180,E1 -14873.461,E2 -14873.461} C_VEL
LIN {X 0,Y 338.084,Z 636.445,A -85,B 0,C 180,E1 -14875.223,E2 -14875.223} C_VEL
LIN {X 0,Y 340.586,Z 624.186,A -85,B 0,C 180,E1 -14876.668,E2 -14876.668} C_VEL
LIN {X 0,Y 343.022,Z 610.814,A -85,B 0,C 180,E1 -14877.948,E2 -14877.948} C_VEL
LIN {X 0,Y 345.024,Z 597.612,A -85,B 0,C 180,E1 -14878.968,E2 -14878.968} C_VEL
LIN {X 0,Y 346.905,Z 583.02,A -85,B 0,C 180,E1 -14879.842,E2 -14879.842} C_VEL
LIN {X 0,Y 348.487,Z 568.066,A -85,B 0,C 180,E1 -14880.486,E2 -14880.486} C_VEL
LIN {X 0,Y 349.521,Z 552.627,A -85,B 0,C 180,E1 -14880.931,E2 -14880.931} C_VEL
LIN {X 0,Y 353.285,Z 442.248,A -85,B 0,C 180,E1 -14883.229,E2 -14883.229} C_VEL
LIN {X 0,Y 350.402,Z 426.875,A -85,B 0,C 180,E1 -14883.968,E2 -14883.968} C_VEL
LIN {X 0,Y 343.727,Z 412.806,A -85,B 0,C 180,E1 -14885.191,E2 -14885.191} C_VEL
LIN {X 0,Y 336.796,Z 399.64,A -85,B 0,C 180,E1 -14886.501,E2 -14886.501} C_VEL
LIN {X 0,Y 332.008,Z 390.9,A -85,B 0,C 180,E1 -14887.459,E2 -14887.459} C_VEL
LIN {X 0,Y 328.889,Z 380.552,A -85,B 0,C 180,E1 -14890.66,E2 -14890.66} C_VEL
LIN {X 0,Y 326.555,Z 373.428,A -85,B 0,C 180,E1 -14893.073,E2 -14893.073} C_VEL
LIN {X 0,Y 326.572,Z 373.433,A -85,B 0,C 180,E1 -14897.029,E2 -14897.029} C_VEL
LIN {X 0,Y 326.581,Z 373.43,A -85,B 0,C 180,E1 -14901.386,E2 -14901.386} C_VEL
LIN {X 0,Y 326.618,Z 373.407,A -85,B 0,C 180,E1 -14904.852,E2 -14904.852} C_VEL
LIN {X 0,Y 326.61,Z 373.415,A -85,B 0,C 180,E1 -14907.456,E2 -14907.456} C_VEL
LIN {X 0,Y 326.617,Z 373.403,A -85,B 0,C 180,E1 -14910.337,E2 -14910.337} C_VEL
LIN {X 0,Y 326.616,Z 373.419,A -85,B 0,C 180,E1 -14913.137,E2 -14913.137} C_VEL
LIN {X 0,Y 326.635,Z 373.424,A -85,B 0,C 180,E1 -14915.87,E2 -14915.87} C_VEL
LIN {X 0,Y 326.66,Z 373.416,A -85,B 0,C 180,E1 -14919.865,E2 -14919.865} C_VEL
LIN {X 0,Y 326.7,Z 373.416,A -85,B 0,C 180,E1 -14922.473,E2 -14922.473} C_VEL
LIN {X 0,Y 326.76,Z 373.408,A -85,B 0,C 180,E1 -14926.315,E2 -14926.315} C_VEL
LIN {X 0,Y 326.784,Z 373.406,A -85,B 0,C 180,E1 -14930.093,E2 -14930.093} C_VEL
LIN {X 0,Y 326.946,Z 373.384,A -85,B 0,C 180,E1 -14933.83,E2 -14933.83} C_VEL
LIN {X 0,Y 327.042,Z 373.372,A -85,B 0,C 180,E1 -14937.537,E2 -14937.537} C_VEL
LIN {X 0,Y 327.048,Z 373.371,A -85,B 0,C 180,E1 -14941.232,E2 -14941.232} C_VEL
LIN {X 0,Y 326.764,Z 373.396,A -85,B 0,C 180,E1 -14943.7,E2 -14943.7} C_VEL
LIN {X 0,Y 326.921,Z 373.381,A -85,B 0,C 180,E1 -14946.542,E2 -14946.542} C_VEL
LIN {X 0,Y 326.806,Z 373.402,A -85,B 0,C 180,E1 -14949.907,E2 -14949.907} C_VEL
LIN {X 0,Y 326.761,Z 373.406,A -85,B 0,C 180,E1 -14953.686,E2 -14953.686} C_VEL
LIN {X 0,Y 326.702,Z 373.409,A -85,B 0,C 180,E1 -14957.528,E2 -14957.528} C_VEL
LIN {X 0,Y 326.66,Z 373.389,A -85,B 0,C 180,E1 -14960.136,E2 -14960.136} C_VEL
LIN {X 0,Y 326.59,Z 373.416,A -85,B 0,C 180,E1 -14964.134,E2 -14964.134} C_VEL
LIN {X 0,Y 326.628,Z 373.424,A -85,B 0,C 180,E1 -14968.254,E2 -14968.254} C_VEL
LIN {X 0,Y 326.577,Z 373.409,A -85,B 0,C 180,E1 -14971.098,E2 -14971.098} C_VEL
LIN {X 0,Y 326.609,Z 373.422,A -85,B 0,C 180,E1 -14974.02,E2 -14974.02} C_VEL
LIN {X 0,Y 326.624,Z 373.425,A -85,B 0,C 180,E1 -14977.238,E2 -14977.238} C_VEL
LIN {X 0,Y 326.617,Z 373.604,A -85,B 0,C 180,E1 -14981.022,E2 -14981.022} C_VEL
LIN {X 0,Y 327.499,Z 376.207,A -85,B 0,C 180,E1 -14981.909,E2 -14981.909} C_VEL
LIN {X 0,Y 329.557,Z 379.728,A -85,B 0,C 180,E1 -14982.333,E2 -14982.333} C_VEL
LIN {X 0,Y 336.412,Z 390.825,A -85,B 0,C 180,E1 -14983.671,E2 -14983.671} C_VEL
LIN {X 0,Y 344.278,Z 404.645,A -85,B 0,C 180,E1 -14985.137,E2 -14985.137} C_VEL
LIN {X 0,Y 352.339,Z 420.778,A -85,B 0,C 180,E1 -14986.588,E2 -14986.588} C_VEL
LIN {X 0,Y 353.875,Z 424.179,A -85,B 0,C 180,E1 -14986.861,E2 -14986.861} C_VEL
LIN {X 0,Y 350.008,Z 527.944,A -85,B 0,C 180,E1 -14988.978,E2 -14988.978} C_VEL
LIN {X 0,Y 349.377,Z 544.583,A -85,B 0,C 180,E1 -14989.411,E2 -14989.411} C_VEL
LIN {X 0,Y 348.158,Z 559.411,A -85,B 0,C 180,E1 -14989.989,E2 -14989.989} C_VEL
LIN {X 0,Y 346.592,Z 574.235,A -85,B 0,C 180,E1 -14990.812,E2 -14990.812} C_VEL
LIN {X 0,Y 344.709,Z 587.292,A -85,B 0,C 180,E1 -14991.735,E2 -14991.735} C_VEL
LIN {X 0,Y 342.781,Z 600.293,A -85,B 0,C 180,E1 -14992.913,E2 -14992.913} C_VEL
LIN {X 0,Y 340.353,Z 613.101,A -85,B 0,C 180,E1 -14994.314,E2 -14994.314} C_VEL
LIN {X 0,Y 337.969,Z 624.587,A -85,B 0,C 180,E1 -14995.843,E2 -14995.843} C_VEL
LIN {X 0,Y 335.4,Z 636.088,A -85,B 0,C 180,E1 -14997.701,E2 -14997.701} C_VEL
LIN {X 0,Y 333.201,Z 645.714,A -85,B 0,C 180,E1 -14999.588,E2 -14999.588} C_VEL
LIN {X 0,Y 330.939,Z 655.096,A -85,B 0,C 180,E1 -15001.802,E2 -15001.802} C_VEL
LIN {X 0,Y 329.03,Z 663.188,A -85,B 0,C 180,E1 -15004.153,E2 -15004.153} C_VEL
LIN {X 0,Y 327.499,Z 669.976,A -85,B 0,C 180,E1 -15006.609,E2 -15006.609} C_VEL
LIN {X 0,Y 326.325,Z 675.534,A -85,B 0,C 180,E1 -15009.185,E2 -15009.185} C_VEL
LIN {X 0,Y 325.593,Z 679.66,A -85,B 0,C 180,E1 -15011.762,E2 -15011.762} C_VEL
LIN {X 0,Y 325.158,Z 681.919,A -85,B 0,C 180,E1 -15013.681,E2 -15013.681} C_VEL
LIN {X 0,Y 324.923,Z 683.829,A -85,B 0,C 180,E1 -15016.236,E2 -15016.236} C_VEL
LIN {X 0,Y 324.767,Z 684.521,A -85,B 0,C 180,E1 -15018.769,E2 -15018.769} C_VEL
LIN {X 0,Y 324.723,Z 684.062,A -85,B 0,C 180,E1 -15021.286,E2 -15021.286} C_VEL
LIN {X 0,Y 324.995,Z 682.147,A -85,B 0,C 180,E1 -15024.133,E2 -15024.133} C_VEL
LIN {X 0,Y 325.123,Z 679.698,A -85,B 0,C 180,E1 -15026.282,E2 -15026.282} C_VEL
LIN {X 0,Y 325.508,Z 675.721,A -85,B 0,C 180,E1 -15028.763,E2 -15028.763} C_VEL
LIN {X 0,Y 326.064,Z 670.433,A -85,B 0,C 180,E1 -15031.235,E2 -15031.235} C_VEL
LIN {X 0,Y 327.049,Z 663.695,A -85,B 0,C 180,E1 -15033.696,E2 -15033.696} C_VEL
LIN {X 0,Y 328.478,Z 655.314,A -85,B 0,C 180,E1 -15036.141,E2 -15036.141} C_VEL
LIN {X 0,Y 330.006,Z 646.396,A -85,B 0,C 180,E1 -15038.265,E2 -15038.265} C_VEL
LIN {X 0,Y 331.86,Z 635.691,A -85,B 0,C 180,E1 -15040.37,E2 -15040.37} C_VEL
LIN {X 0,Y 333.964,Z 623.65,A -85,B 0,C 180,E1 -15042.303,E2 -15042.303} C_VEL
LIN {X 0,Y 335.785,Z 611.429,A -85,B 0,C 180,E1 -15043.928,E2 -15043.928} C_VEL
LIN {X 0,Y 337.771,Z 597.919,A -85,B 0,C 180,E1 -15045.384,E2 -15045.384} C_VEL
LIN {X 0,Y 339.402,Z 584.699,A -85,B 0,C 180,E1 -15046.542,E2 -15046.542} C_VEL
LIN {X 0,Y 340.932,Z 570.092,A -85,B 0,C 180,E1 -15047.547,E2 -15047.547} C_VEL
LIN {X 0,Y 342.164,Z 555.607,A -85,B 0,C 180,E1 -15048.293,E2 -15048.293} C_VEL
LIN {X 0,Y 343.004,Z 539.849,A -85,B 0,C 180,E1 -15048.866,E2 -15048.866} C_VEL
LIN {X 0,Y 345.868,Z 441.916,A -85,B 0,C 180,E1 -15050.912,E2 -15050.912} C_VEL
LIN {X 0,Y 345.328,Z 436.126,A -85,B 0,C 180,E1 -15051.093,E2 -15051.093} C_VEL
LIN {X 0,Y 343.915,Z 430.556,A -85,B 0,C 180,E1 -15051.348,E2 -15051.348} C_VEL
LIN {X 0,Y 337.12,Z 412.652,A -85,B 0,C 180,E1 -15052.394,E2 -15052.394} C_VEL
LIN {X 0,Y 329.643,Z 395.538,A -85,B 0,C 180,E1 -15053.541,E2 -15053.541} C_VEL
LIN {X 0,Y 321.379,Z 378.553,A -85,B 0,C 180,E1 -15054.836,E2 -15054.836} C_VEL
LIN {X 0,Y 319.725,Z 375.151,A -85,B 0,C 180,E1 -15055.151,E2 -15055.151} C_VEL
LIN {X 0,Y 319.582,Z 374.3,A -85,B 0,C 180,E1 -15055.439,E2 -15055.439} C_VEL
LIN {X 0,Y 319.547,Z 374.302,A -85,B 0,C 180,E1 -15058.938,E2 -15058.938} C_VEL
LIN {X 0,Y 319.529,Z 374.302,A -85,B 0,C 180,E1 -15061.862,E2 -15061.862} C_VEL
LIN {X 0,Y 319.583,Z 374.294,A -85,B 0,C 180,E1 -15065.542,E2 -15065.542} C_VEL
LIN {X 0,Y 319.531,Z 374.298,A -85,B 0,C 180,E1 -15069.662,E2 -15069.662} C_VEL
LIN {X 0,Y 319.524,Z 374.31,A -85,B 0,C 180,E1 -15073.46,E2 -15073.46} C_VEL
LIN {X 0,Y 319.555,Z 374.291,A -85,B 0,C 180,E1 -15077.016,E2 -15077.016} C_VEL
LIN {X 0,Y 319.517,Z 374.304,A -85,B 0,C 180,E1 -15080.366,E2 -15080.366} C_VEL
LIN {X 0,Y 319.581,Z 374.299,A -85,B 0,C 180,E1 -15084.457,E2 -15084.457} C_VEL
LIN {X 0,Y 319.527,Z 374.31,A -85,B 0,C 180,E1 -15088.137,E2 -15088.137} C_VEL
LIN {X 0,Y 319.572,Z 374.276,A -85,B 0,C 180,E1 -15091.604,E2 -15091.604} C_VEL
LIN {X 0,Y 319.53,Z 374.27,A -85,B 0,C 180,E1 -15095.297,E2 -15095.297} C_VEL
LIN {X 0,Y 319.569,Z 374.301,A -85,B 0,C 180,E1 -15098.045,E2 -15098.045} C_VEL
LIN {X 0,Y 319.627,Z 374.28,A -85,B 0,C 180,E1 -15102.071,E2 -15102.071} C_VEL
LIN {X 0,Y 319.735,Z 374.279,A -85,B 0,C 180,E1 -15106.007,E2 -15106.007} C_VEL
LIN {X 0,Y 319.738,Z 374.271,A -85,B 0,C 180,E1 -15109.872,E2 -15109.872} C_VEL
LIN {X 0,Y 319.9,Z 374.25,A -85,B 0,C 180,E1 -15113.693,E2 -15113.693} C_VEL
LIN {X 0,Y 319.958,Z 374.252,A -85,B 0,C 180,E1 -15117.482,E2 -15117.482} C_VEL
LIN {X 0,Y 320.003,Z 374.234,A -85,B 0,C 180,E1 -15121.258,E2 -15121.258} C_VEL
LIN {X 0,Y 319.718,Z 374.282,A -85,B 0,C 180,E1 -15123.781,E2 -15123.781} C_VEL
LIN {X 0,Y 319.902,Z 374.256,A -85,B 0,C 180,E1 -15126.306,E2 -15126.306} C_VEL
LIN {X 0,Y 319.737,Z 374.28,A -85,B 0,C 180,E1 -15130.127,E2 -15130.127} C_VEL
LIN {X 0,Y 319.71,Z 374.277,A -85,B 0,C 180,E1 -15133.993,E2 -15133.993} C_VEL
LIN {X 0,Y 319.617,Z 374.286,A -85,B 0,C 180,E1 -15137.929,E2 -15137.929} C_VEL
LIN {X 0,Y 319.607,Z 374.293,A -85,B 0,C 180,E1 -15140.599,E2 -15140.599} C_VEL
LIN {X 0,Y 319.562,Z 374.297,A -85,B 0,C 180,E1 -15143.32,E2 -15143.32} C_VEL
LIN {X 0,Y 319.57,Z 374.295,A -85,B 0,C 180,E1 -15146.093,E2 -15146.093} C_VEL
LIN {X 0,Y 319.543,Z 374.305,A -85,B 0,C 180,E1 -15148.938,E2 -15148.938} C_VEL
LIN {X 0,Y 319.524,Z 374.308,A -85,B 0,C 180,E1 -15151.862,E2 -15151.862} C_VEL
LIN {X 0,Y 319.579,Z 374.3,A -85,B 0,C 180,E1 -15155.542,E2 -15155.542} C_VEL
LIN {X 0,Y 319.527,Z 374.295,A -85,B 0,C 180,E1 -15159.661,E2 -15159.661} C_VEL
LIN {X 0,Y 319.519,Z 374.311,A -85,B 0,C 180,E1 -15163.46,E2 -15163.46} C_VEL
LIN {X 0,Y 319.551,Z 374.308,A -85,B 0,C 180,E1 -15167.016,E2 -15167.016} C_VEL
LIN {X 0,Y 319.544,Z 374.339,A -85,B 0,C 180,E1 -15170.768,E2 -15170.768} C_VEL
LIN {X 0,Y 322.76,Z 386.19,A -85,B 0,C 180,E1 -15173.99,E2 -15173.99} C_VEL
LIN {X 0,Y 324.1,Z 391.614,A -85,B 0,C 180,E1 -15175.386,E2 -15175.386} C_VEL
LIN {X 0,Y 334.313,Z 415.209,A -85,B 0,C 180,E1 -15176.998,E2 -15176.998} C_VEL
LIN {X 0,Y 336.192,Z 420.398,A -85,B 0,C 180,E1 -15177.302,E2 -15177.302} C_VEL
LIN {X 0,Y 339.739,Z 442.48,A -85,B 0,C 180,E1 -15178.155,E2 -15178.155} C_VEL
LIN {X 0,Y 336.308,Z 558.871,A -85,B 0,C 180,E1 -15180.63,E2 -15180.63} C_VEL
LIN {X 0,Y 335.282,Z 574.096,A -85,B 0,C 180,E1 -15181.176,E2 -15181.176} C_VEL
LIN {X 0,Y 333.857,Z 588.299,A -85,B 0,C 180,E1 -15181.9,E2 -15181.9} C_VEL
LIN {X 0,Y 332.154,Z 603.488,A -85,B 0,C 180,E1 -15182.947,E2 -15182.947} C_VEL
LIN {X 0,Y 330.253,Z 617,A -85,B 0,C 180,E1 -15184.135,E2 -15184.135} C_VEL
LIN {X 0,Y 328.357,Z 629.519,A -85,B 0,C 180,E1 -15185.5,E2 -15185.5} C_VEL
LIN {X 0,Y 326.325,Z 641.147,A -85,B 0,C 180,E1 -15187.023,E2 -15187.023} C_VEL
LIN {X 0,Y 324.482,Z 652.278,A -85,B 0,C 180,E1 -15188.783,E2 -15188.783} C_VEL
LIN {X 0,Y 322.855,Z 661.989,A -85,B 0,C 180,E1 -15190.612,E2 -15190.612} C_VEL
LIN {X 0,Y 321.133,Z 671.763,A -85,B 0,C 180,E1 -15192.816,E2 -15192.816} C_VEL
LIN {X 0,Y 320.032,Z 678.856,A -85,B 0,C 180,E1 -15194.721,E2 -15194.721} C_VEL
LIN {X 0,Y 318.97,Z 686.647,A -85,B 0,C 180,E1 -15197.271,E2 -15197.271} C_VEL
LIN {X 0,Y 318.265,Z 692.824,A -85,B 0,C 180,E1 -15199.825,E2 -15199.825} C_VEL
LIN {X 0,Y 317.933,Z 697.564,A -85,B 0,C 180,E1 -15202.378,E2 -15202.378} C_VEL
LIN {X 0,Y 317.78,Z 700.989,A -85,B 0,C 180,E1 -15204.925,E2 -15204.925} C_VEL
LIN {X 0,Y 317.771,Z 703.186,A -85,B 0,C 180,E1 -15207.465,E2 -15207.465} C_VEL
LIN {X 0,Y 317.797,Z 704.214,A -85,B 0,C 180,E1 -15210,E2 -15210} C_VEL
LIN {X 0,Y 317.758,Z 704.099,A -85,B 0,C 180,E1 -15212.535,E2 -15212.535} C_VEL
LIN {X 0,Y 317.764,Z 702.794,A -85,B 0,C 180,E1 -15215.075,E2 -15215.075} C_VEL
LIN {X 0,Y 317.918,Z 700.324,A -85,B 0,C 180,E1 -15217.622,E2 -15217.622} C_VEL
LIN {X 0,Y 318.356,Z 696.668,A -85,B 0,C 180,E1 -15220.172,E2 -15220.172} C_VEL
LIN {X 0,Y 319.189,Z 691.743,A -85,B 0,C 180,E1 -15222.72,E2 -15222.72} C_VEL
LIN {X 0,Y 320.329,Z 685.424,A -85,B 0,C 180,E1 -15225.265,E2 -15225.265} C_VEL
LIN {X 0,Y 322.13,Z 677.54,A -85,B 0,C 180,E1 -15227.785,E2 -15227.785} C_VEL
LIN {X 0,Y 324.103,Z 669.185,A -85,B 0,C 180,E1 -15229.97,E2 -15229.97} C_VEL
LIN {X 0,Y 326.471,Z 659.434,A -85,B 0,C 180,E1 -15232.074,E2 -15232.074} C_VEL
LIN {X 0,Y 328.897,Z 648.947,A -85,B 0,C 180,E1 -15233.954,E2 -15233.954} C_VEL
LIN {X 0,Y 331.685,Z 636.774,A -85,B 0,C 180,E1 -15235.745,E2 -15235.745} C_VEL
LIN {X 0,Y 334.558,Z 623.252,A -85,B 0,C 180,E1 -15237.356,E2 -15237.356} C_VEL
LIN {X 0,Y 337.039,Z 609.752,A -85,B 0,C 180,E1 -15238.659,E2 -15238.659} C_VEL
LIN {X 0,Y 339.14,Z 596.661,A -85,B 0,C 180,E1 -15239.667,E2 -15239.667} C_VEL
LIN {X 0,Y 340.994,Z 582.79,A -85,B 0,C 180,E1 -15240.499,E2 -15240.499} C_VEL
LIN {X 0,Y 342.614,Z 567.846,A -85,B 0,C 180,E1 -15241.152,E2 -15241.152} C_VEL
LIN {X 0,Y 343.702,Z 552.413,A -85,B 0,C 180,E1 -15241.6,E2 -15241.6} C_VEL
LIN {X 0,Y 347.503,Z 443.01,A -85,B 0,C 180,E1 -15243.92,E2 -15243.92} C_VEL
LIN {X 0,Y 345.121,Z 430.026,A -85,B 0,C 180,E1 -15244.558,E2 -15244.558} C_VEL
LIN {X 0,Y 337.927,Z 414.862,A -85,B 0,C 180,E1 -15245.927,E2 -15245.927} C_VEL
LIN {X 0,Y 331.128,Z 402.134,A -85,B 0,C 180,E1 -15247.259,E2 -15247.259} C_VEL
LIN {X 0,Y 324.648,Z 390.566,A -85,B 0,C 180,E1 -15248.615,E2 -15248.615} C_VEL
LIN {X 0,Y 321.459,Z 380.219,A -85,B 0,C 180,E1 -15251.984,E2 -15251.984} C_VEL
LIN {X 0,Y 319.484,Z 374.312,A -85,B 0,C 180,E1 -15254.111,E2 -15254.111} C_VEL
LIN {X 0,Y 319.551,Z 374.307,A -85,B 0,C 180,E1 -15257.016,E2 -15257.016} C_VEL
LIN {X 0,Y 319.543,Z 374.303,A -85,B 0,C 180,E1 -15260.371,E2 -15260.371} C_VEL
LIN {X 0,Y 319.578,Z 374.28,A -85,B 0,C 180,E1 -15264.458,E2 -15264.458} C_VEL
LIN {X 0,Y 319.525,Z 374.284,A -85,B 0,C 180,E1 -15268.138,E2 -15268.138} C_VEL
LIN {X 0,Y 319.588,Z 374.297,A -85,B 0,C 180,E1 -15271.598,E2 -15271.598} C_VEL
LIN {X 0,Y 319.576,Z 374.302,A -85,B 0,C 180,E1 -15275.302,E2 -15275.302} C_VEL
LIN {X 0,Y 319.59,Z 374.297,A -85,B 0,C 180,E1 -15278.048,E2 -15278.048} C_VEL
LIN {X 0,Y 319.689,Z 374.282,A -85,B 0,C 180,E1 -15280.963,E2 -15280.963} C_VEL
LIN {X 0,Y 319.732,Z 374.281,A -85,B 0,C 180,E1 -15285.276,E2 -15285.276} C_VEL
LIN {X 0,Y 319.716,Z 374.279,A -85,B 0,C 180,E1 -15288.59,E2 -15288.59} C_VEL
LIN {X 0,Y 319.854,Z 374.261,A -85,B 0,C 180,E1 -15292.425,E2 -15292.425} C_VEL
LIN {X 0,Y 319.729,Z 374.275,A -85,B 0,C 180,E1 -15294.956,E2 -15294.956} C_VEL
LIN {X 0,Y 319.985,Z 374.251,A -85,B 0,C 180,E1 -15297.483,E2 -15297.483} C_VEL
LIN {X 0,Y 320.015,Z 374.247,A -85,B 0,C 180,E1 -15301.259,E2 -15301.259} C_VEL
LIN {X 0,Y 319.726,Z 374.284,A -85,B 0,C 180,E1 -15305.045,E2 -15305.045} C_VEL
LIN {X 0,Y 319.855,Z 374.257,A -85,B 0,C 180,E1 -15307.576,E2 -15307.576} C_VEL
LIN {X 0,Y 319.725,Z 374.276,A -85,B 0,C 180,E1 -15311.411,E2 -15311.411} C_VEL
LIN {X 0,Y 319.702,Z 374.282,A -85,B 0,C 180,E1 -15315.296,E2 -15315.296} C_VEL
LIN {X 0,Y 319.654,Z 374.261,A -85,B 0,C 180,E1 -15319.257,E2 -15319.257} C_VEL
LIN {X 0,Y 319.536,Z 374.306,A -85,B 0,C 180,E1 -15323.323,E2 -15323.323} C_VEL
LIN {X 0,Y 319.558,Z 374.277,A -85,B 0,C 180,E1 -15326.096,E2 -15326.096} C_VEL
LIN {X 0,Y 319.56,Z 374.303,A -85,B 0,C 180,E1 -15328.937,E2 -15328.937} C_VEL
LIN {X 0,Y 319.527,Z 374.291,A -85,B 0,C 180,E1 -15331.863,E2 -15331.863} C_VEL
LIN {X 0,Y 319.58,Z 374.283,A -85,B 0,C 180,E1 -15335.543,E2 -15335.543} C_VEL
LIN {X 0,Y 319.526,Z 374.304,A -85,B 0,C 180,E1 -15338.016,E2 -15338.016} C_VEL
LIN {X 0,Y 319.534,Z 374.423,A -85,B 0,C 180,E1 -15340.001,E2 -15340.001} C_VEL
LIN {X 0,Y 320.18,Z 376.485,A -85,B 0,C 180,E1 -15340.718,E2 -15340.718} C_VEL
LIN {X 0,Y 322.848,Z 380.624,A -85,B 0,C 180,E1 -15341.289,E2 -15341.289} C_VEL
LIN {X 0,Y 331.983,Z 395.435,A -85,B 0,C 180,E1 -15343.149,E2 -15343.149} C_VEL
LIN {X 0,Y 339.588,Z 409.008,A -85,B 0,C 180,E1 -15344.615,E2 -15344.615} C_VEL
LIN {X 0,Y 346.61,Z 423.098,A -85,B 0,C 180,E1 -15345.924,E2 -15345.924} C_VEL
LIN {X 0,Y 348.109,Z 426.329,A -85,B 0,C 180,E1 -15346.199,E2 -15346.199} C_VEL
LIN {X 0,Y 344.411,Z 523.359,A -85,B 0,C 180,E1 -15348.212,E2 -15348.212} C_VEL
LIN {X 0,Y 343.604,Z 542.869,A -85,B 0,C 180,E1 -15348.679,E2 -15348.679} C_VEL
LIN {X 0,Y 342.392,Z 558.235,A -85,B 0,C 180,E1 -15349.264,E2 -15349.264} C_VEL
LIN {X 0,Y 340.845,Z 572.933,A -85,B 0,C 180,E1 -15350.068,E2 -15350.068} C_VEL
LIN {X 0,Y 338.943,Z 585.856,A -85,B 0,C 180,E1 -15350.963,E2 -15350.963} C_VEL
LIN {X 0,Y 336.806,Z 599.754,A -85,B 0,C 180,E1 -15352.216,E2 -15352.216} C_VEL
LIN {X 0,Y 334.384,Z 612.227,A -85,B 0,C 180,E1 -15353.582,E2 -15353.582} C_VEL
LIN {X 0,Y 331.886,Z 623.801,A -85,B 0,C 180,E1 -15355.128,E2 -15355.128} C_VEL
LIN {X 0,Y 329.162,Z 635.474,A -85,B 0,C 180,E1 -15357.012,E2 -15357.012} C_VEL
LIN {X 0,Y 326.836,Z 645.227,A -85,B 0,C 180,E1 -15358.931,E2 -15358.931} C_VEL
LIN {X 0,Y 324.411,Z 654.731,A -85,B 0,C 180,E1 -15361.182,E2 -15361.182} C_VEL
LIN {X 0,Y 322.313,Z 663.277,A -85,B 0,C 180,E1 -15363.69,E2 -15363.69} C_VEL
LIN {X 0,Y 320.713,Z 669.815,A -85,B 0,C 180,E1 -15366.084,E2 -15366.084} C_VEL
LIN {X 0,Y 319.415,Z 675.46,A -85,B 0,C 180,E1 -15368.713,E2 -15368.713} C_VEL
LIN {X 0,Y 318.558,Z 679.966,A -85,B 0,C 180,E1 -15371.564,E2 -15371.564} C_VEL
LIN {X 0,Y 318.152,Z 682,A -85,B 0,C 180,E1 -15373.311,E2 -15373.311} C_VEL
LIN {X 0,Y 317.856,Z 683.956,A -85,B 0,C 180,E1 -15375.924,E2 -15375.924} C_VEL
LIN {X 0,Y 317.702,Z 684.722,A -85,B 0,C 180,E1 -15378.516,E2 -15378.516} C_VEL
LIN {X 0,Y 317.623,Z 684.339,A -85,B 0,C 180,E1 -15381.09,E2 -15381.09} C_VEL
LIN {X 0,Y 317.846,Z 682.809,A -85,B 0,C 180,E1 -15383.653,E2 -15383.653} C_VEL
LIN {X 0,Y 318.037,Z 680.126,A -85,B 0,C 180,E1 -15386.199,E2 -15386.199} C_VEL
LIN {X 0,Y 318.433,Z 676.211,A -85,B 0,C 180,E1 -15388.735,E2 -15388.735} C_VEL
LIN {X 0,Y 318.997,Z 670.985,A -85,B 0,C 180,E1 -15391.262,E2 -15391.262} C_VEL
LIN {X 0,Y 319.986,Z 664.335,A -85,B 0,C 180,E1 -15393.778,E2 -15393.778} C_VEL
LIN {X 0,Y 321.45,Z 656.058,A -85,B 0,C 180,E1 -15396.276,E2 -15396.276} C_VEL
LIN {X 0,Y 323.032,Z 647.235,A -85,B 0,C 180,E1 -15398.445,E2 -15398.445} C_VEL
LIN {X 0,Y 324.646,Z 638.264,A -85,B 0,C 180,E1 -15400.288,E2 -15400.288} C_VEL
LIN {X 0,Y 326.591,Z 627.693,A -85,B 0,C 180,E1 -15402.112,E2 -15402.112} C_VEL
LIN {X 0,Y 328.635,Z 615.056,A -85,B 0,C 180,E1 -15403.921,E2 -15403.921} C_VEL
LIN {X 0,Y 330.576,Z 602.315,A -85,B 0,C 180,E1 -15405.412,E2 -15405.412} C_VEL
LIN {X 0,Y 332.507,Z 588.261,A -85,B 0,C 180,E1 -15406.737,E2 -15406.737} C_VEL
LIN {X 0,Y 334.043,Z 574.598,A -85,B 0,C 180,E1 -15407.762,E2 -15407.762} C_VEL
LIN {X 0,Y 335.351,Z 560.108,A -85,B 0,C 180,E1 -15408.599,E2 -15408.599} C_VEL
LIN {X 0,Y 336.331,Z 545.324,A -85,B 0,C 180,E1 -15409.215,E2 -15409.215} C_VEL
LIN {X 0,Y 337.066,Z 528.495,A -85,B 0,C 180,E1 -15409.653,E2 -15409.653} C_VEL
LIN {X 0,Y 340.145,Z 420.145,A -85,B 0,C 180,E1 -15411.933,E2 -15411.933} C_VEL
LIN {X 0,Y 337.12,Z 412.652,A -85,B 0,C 180,E1 -15412.394,E2 -15412.394} C_VEL
LIN {X 0,Y 334.768,Z 407.679,A -85,B 0,C 180,E1 -15412.738,E2 -15412.738} C_VEL
LIN {X 0,Y 331.528,Z 403.379,A -85,B 0,C 180,E1 -15413.159,E2 -15413.159} C_VEL
LIN {X 0,Y 321.834,Z 392.835,A -85,B 0,C 180,E1 -15414.42,E2 -15414.42} C_VEL
LIN {X 0,Y 319.8,Z 389.81,A -85,B 0,C 180,E1 -15414.717,E2 -15414.717} C_VEL
LIN {X 0,Y 313.81,Z 378.444,A -85,B 0,C 180,E1 -15415.684,E2 -15415.684} C_VEL
LIN {X 0,Y 312.637,Z 375.885,A -85,B 0,C 180,E1 -15415.887,E2 -15415.887} C_VEL
LIN {X 0,Y 312.513,Z 375.183,A -85,B 0,C 180,E1 -15416.069,E2 -15416.069} C_VEL
LIN {X 0,Y 312.5,Z 375.177,A -85,B 0,C 180,E1 -15419.655,E2 -15419.655} C_VEL
LIN {X 0,Y 312.524,Z 375.177,A -85,B 0,C 180,E1 -15423.689,E2 -15423.689} C_VEL
LIN {X 0,Y 312.518,Z 375.176,A -85,B 0,C 180,E1 -15427.386,E2 -15427.386} C_VEL
LIN {X 0,Y 312.444,Z 375.175,A -85,B 0,C 180,E1 -15430.717,E2 -15430.717} C_VEL
LIN {X 0,Y 312.454,Z 375.184,A -85,B 0,C 180,E1 -15434.209,E2 -15434.209} C_VEL
LIN {X 0,Y 312.459,Z 375.185,A -85,B 0,C 180,E1 -15437.924,E2 -15437.924} C_VEL
LIN {X 0,Y 312.479,Z 375.181,A -85,B 0,C 180,E1 -15441.924,E2 -15441.924} C_VEL
LIN {X 0,Y 312.533,Z 375.178,A -85,B 0,C 180,E1 -15444.22,E2 -15444.22} C_VEL
LIN {X 0,Y 312.504,Z 375.181,A -85,B 0,C 180,E1 -15447.333,E2 -15447.333} C_VEL
LIN {X 0,Y 312.507,Z 375.159,A -85,B 0,C 180,E1 -15451.292,E2 -15451.292} C_VEL
LIN {X 0,Y 312.519,Z 375.134,A -85,B 0,C 180,E1 -15454.704,E2 -15454.704} C_VEL
LIN {X 0,Y 312.543,Z 375.169,A -85,B 0,C 180,E1 -15457.525,E2 -15457.525} C_VEL
LIN {X 0,Y 312.585,Z 375.16,A -85,B 0,C 180,E1 -15461.652,E2 -15461.652} C_VEL
LIN {X 0,Y 312.689,Z 375.16,A -85,B 0,C 180,E1 -15465.685,E2 -15465.685} C_VEL
LIN {X 0,Y 312.688,Z 375.146,A -85,B 0,C 180,E1 -15469.641,E2 -15469.641} C_VEL
LIN {X 0,Y 312.798,Z 375.142,A -85,B 0,C 180,E1 -15472.252,E2 -15472.252} C_VEL
LIN {X 0,Y 312.69,Z 375.142,A -85,B 0,C 180,E1 -15474.841,E2 -15474.841} C_VEL
LIN {X 0,Y 312.982,Z 375.121,A -85,B 0,C 180,E1 -15478.713,E2 -15478.713} C_VEL
LIN {X 0,Y 312.925,Z 375.12,A -85,B 0,C 180,E1 -15482.574,E2 -15482.574} C_VEL
LIN {X 0,Y 312.844,Z 375.135,A -85,B 0,C 180,E1 -15486.449,E2 -15486.449} C_VEL
LIN {X 0,Y 312.752,Z 375.144,A -85,B 0,C 180,E1 -15489.05,E2 -15489.05} C_VEL
LIN {X 0,Y 312.626,Z 375.155,A -85,B 0,C 180,E1 -15492.991,E2 -15492.991} C_VEL
LIN {X 0,Y 312.576,Z 375.173,A -85,B 0,C 180,E1 -15495.652,E2 -15495.652} C_VEL
LIN {X 0,Y 312.578,Z 375.171,A -85,B 0,C 180,E1 -15499.709,E2 -15499.709} C_VEL
LIN {X 0,Y 312.541,Z 375.168,A -85,B 0,C 180,E1 -15502.786,E2 -15502.786} C_VEL
LIN {X 0,Y 312.53,Z 375.173,A -85,B 0,C 180,E1 -15505.907,E2 -15505.907} C_VEL
LIN {X 0,Y 312.496,Z 375.18,A -85,B 0,C 180,E1 -15509.655,E2 -15509.655} C_VEL
LIN {X 0,Y 312.519,Z 375.18,A -85,B 0,C 180,E1 -15513.688,E2 -15513.688} C_VEL
LIN {X 0,Y 312.51,Z 375.184,A -85,B 0,C 180,E1 -15517.387,E2 -15517.387} C_VEL
LIN {X 0,Y 312.44,Z 375.186,A -85,B 0,C 180,E1 -15520.716,E2 -15520.716} C_VEL
LIN {X 0,Y 312.45,Z 375.189,A -85,B 0,C 180,E1 -15524.209,E2 -15524.209} C_VEL
LIN {X 0,Y 312.454,Z 375.192,A -85,B 0,C 180,E1 -15527.924,E2 -15527.924} C_VEL
LIN {X 0,Y 312.494,Z 375.269,A -85,B 0,C 180,E1 -15530.139,E2 -15530.139} C_VEL
LIN {X 0,Y 314.979,Z 384.148,A -85,B 0,C 180,E1 -15532.66,E2 -15532.66} C_VEL
LIN {X 0,Y 316.912,Z 391.579,A -85,B 0,C 180,E1 -15534.609,E2 -15534.609} C_VEL
LIN {X 0,Y 327.469,Z 415.633,A -85,B 0,C 180,E1 -15536.336,E2 -15536.336} C_VEL
LIN {X 0,Y 330.266,Z 423.003,A -85,B 0,C 180,E1 -15536.795,E2 -15536.795} C_VEL
LIN {X 0,Y 333.452,Z 442.42,A -85,B 0,C 180,E1 -15537.574,E2 -15537.574} C_VEL
LIN {X 0,Y 330.007,Z 557.397,A -85,B 0,C 180,E1 -15540.057,E2 -15540.057} C_VEL
LIN {X 0,Y 328.938,Z 573.074,A -85,B 0,C 180,E1 -15540.61,E2 -15540.61} C_VEL
LIN {X 0,Y 327.398,Z 588.122,A -85,B 0,C 180,E1 -15541.382,E2 -15541.382} C_VEL
LIN {X 0,Y 325.672,Z 602.853,A -85,B 0,C 180,E1 -15542.41,E2 -15542.41} C_VEL
LIN {X 0,Y 323.564,Z 617.577,A -85,B 0,C 180,E1 -15543.733,E2 -15543.733} C_VEL
LIN {X 0,Y 321.387,Z 631.222,A -85,B 0,C 180,E1 -15545.278,E2 -15545.278} C_VEL
LIN {X 0,Y 319.316,Z 642.573,A -85,B 0,C 180,E1 -15546.832,E2 -15546.832} C_VEL
LIN {X 0,Y 317.344,Z 654.191,A -85,B 0,C 180,E1 -15548.765,E2 -15548.765} C_VEL
LIN {X 0,Y 315.488,Z 664.421,A -85,B 0,C 180,E1 -15550.817,E2 -15550.817} C_VEL
LIN {X 0,Y 313.842,Z 673.746,A -85,B 0,C 180,E1 -15553.075,E2 -15553.075} C_VEL
LIN {X 0,Y 312.696,Z 680.745,A -85,B 0,C 180,E1 -15555.114,E2 -15555.114} C_VEL
LIN {X 0,Y 311.75,Z 687.879,A -85,B 0,C 180,E1 -15557.633,E2 -15557.633} C_VEL
LIN {X 0,Y 311.096,Z 693.737,A -85,B 0,C 180,E1 -15560.245,E2 -15560.245} C_VEL
LIN {X 0,Y 310.867,Z 697.22,A -85,B 0,C 180,E1 -15562.204,E2 -15562.204} C_VEL
LIN {X 0,Y 310.687,Z 700.685,A -85,B 0,C 180,E1 -15564.808,E2 -15564.808} C_VEL
LIN {X 0,Y 310.693,Z 702.922,A -85,B 0,C 180,E1 -15567.407,E2 -15567.407} C_VEL
LIN {X 0,Y 310.707,Z 703.986,A -85,B 0,C 180,E1 -15570,E2 -15570} C_VEL
LIN {X 0,Y 310.679,Z 703.903,A -85,B 0,C 180,E1 -15572.593,E2 -15572.593} C_VEL
LIN {X 0,Y 310.687,Z 702.378,A -85,B 0,C 180,E1 -15575.55,E2 -15575.55} C_VEL
LIN {X 0,Y 310.835,Z 700.189,A -85,B 0,C 180,E1 -15577.797,E2 -15577.797} C_VEL
LIN {X 0,Y 311.314,Z 696.574,A -85,B 0,C 180,E1 -15580.405,E2 -15580.405} C_VEL
LIN {X 0,Y 312.215,Z 691.693,A -85,B 0,C 180,E1 -15583.009,E2 -15583.009} C_VEL
LIN {X 0,Y 313.433,Z 685.42,A -85,B 0,C 180,E1 -15585.609,E2 -15585.609} C_VEL
LIN {X 0,Y 315.34,Z 677.587,A -85,B 0,C 180,E1 -15588.181,E2 -15588.181} C_VEL
LIN {X 0,Y 317.414,Z 669.288,A -85,B 0,C 180,E1 -15590.41,E2 -15590.41} C_VEL
LIN {X 0,Y 319.733,Z 660.132,A -85,B 0,C 180,E1 -15592.445,E2 -15592.445} C_VEL
LIN {X 0,Y 322.412,Z 649.168,A -85,B 0,C 180,E1 -15594.467,E2 -15594.467} C_VEL
LIN {X 0,Y 325.314,Z 637.095,A -85,B 0,C 180,E1 -15596.288,E2 -15596.288} C_VEL
LIN {X 0,Y 328.29,Z 623.726,A -85,B 0,C 180,E1 -15597.924,E2 -15597.924} C_VEL
LIN {X 0,Y 330.86,Z 610.364,A -85,B 0,C 180,E1 -15599.246,E2 -15599.246} C_VEL
LIN {X 0,Y 333.359,Z 595.587,A -85,B 0,C 180,E1 -15600.396,E2 -15600.396} C_VEL
LIN {X 0,Y 335.309,Z 581.284,A -85,B 0,C 180,E1 -15601.249,E2 -15601.249} C_VEL
LIN {X 0,Y 336.968,Z 565.818,A -85,B 0,C 180,E1 -15601.91,E2 -15601.91} C_VEL
LIN {X 0,Y 337.988,Z 550.731,A -85,B 0,C 180,E1 -15602.329,E2 -15602.329} C_VEL
LIN {X 0,Y 341.847,Z 444.422,A -85,B 0,C 180,E1 -15604.608,E2 -15604.608} C_VEL
LIN {X 0,Y 339.781,Z 433.072,A -85,B 0,C 180,E1 -15605.183,E2 -15605.183} C_VEL
LIN {X 0,Y 332.491,Z 417.586,A -85,B 0,C 180,E1 -15606.625,E2 -15606.625} C_VEL
LIN {X 0,Y 325.396,Z 404.363,A -85,B 0,C 180,E1 -15608.072,E2 -15608.072} C_VEL
LIN {X 0,Y 319.792,Z 394.675,A -85,B 0,C 180,E1 -15609.265,E2 -15609.265} C_VEL
LIN {X 0,Y 317.281,Z 390.161,A -85,B 0,C 180,E1 -15609.87,E2 -15609.87} C_VEL
LIN {X 0,Y 314.074,Z 380.077,A -85,B 0,C 180,E1 -15613.345,E2 -15613.345} C_VEL
LIN {X 0,Y 312.469,Z 375.19,A -85,B 0,C 180,E1 -15615.23,E2 -15615.23} C_VEL
LIN {X 0,Y 312.454,Z 375.187,A -85,B 0,C 180,E1 -15617.925,E2 -15617.925} C_VEL
LIN {X 0,Y 312.483,Z 375.181,A -85,B 0,C 180,E1 -15621.923,E2 -15621.923} C_VEL
LIN {X 0,Y 312.53,Z 375.156,A -85,B 0,C 180,E1 -15624.221,E2 -15624.221} C_VEL
LIN {X 0,Y 312.501,Z 375.172,A -85,B 0,C 180,E1 -15627.334,E2 -15627.334} C_VEL
LIN {X 0,Y 312.519,Z 375.174,A -85,B 0,C 180,E1 -15631.288,E2 -15631.288} C_VEL
LIN {X 0,Y 312.548,Z 375.175,A -85,B 0,C 180,E1 -15634.708,E2 -15634.708} C_VEL
LIN {X 0,Y 312.583,Z 375.167,A -85,B 0,C 180,E1 -15637.529,E2 -15637.529} C_VEL
LIN {X 0,Y 312.639,Z 375.164,A -85,B 0,C 180,E1 -15641.657,E2 -15641.657} C_VEL
LIN {X 0,Y 312.695,Z 375.158,A -85,B 0,C 180,E1 -15645.687,E2 -15645.687} C_VEL
LIN {X 0,Y 312.686,Z 375.16,A -85,B 0,C 180,E1 -15649.642,E2 -15649.642} C_VEL
LIN {X 0,Y 312.797,Z 375.138,A -85,B 0,C 180,E1 -15652.253,E2 -15652.253} C_VEL
LIN {X 0,Y 312.698,Z 375.152,A -85,B 0,C 180,E1 -15654.843,E2 -15654.843} C_VEL
LIN {X 0,Y 312.932,Z 375.129,A -85,B 0,C 180,E1 -15657.426,E2 -15657.426} C_VEL
LIN {X 0,Y 312.982,Z 375.123,A -85,B 0,C 180,E1 -15661.287,E2 -15661.287} C_VEL
LIN {X 0,Y 312.696,Z 375.16,A -85,B 0,C 180,E1 -15665.159,E2 -15665.159} C_VEL
LIN {X 0,Y 312.798,Z 375.137,A -85,B 0,C 180,E1 -15667.748,E2 -15667.748} C_VEL
LIN {X 0,Y 312.671,Z 375.155,A -85,B 0,C 180,E1 -15671.672,E2 -15671.672} C_VEL
LIN {X 0,Y 312.702,Z 375.151,A -85,B 0,C 180,E1 -15674.888,E2 -15674.888} C_VEL
LIN {X 0,Y 312.611,Z 375.137,A -85,B 0,C 180,E1 -15679.226,E2 -15679.226} C_VEL
LIN {X 0,Y 312.518,Z 375.183,A -85,B 0,C 180,E1 -15682.776,E2 -15682.776} C_VEL
LIN {X 0,Y 312.496,Z 375.161,A -85,B 0,C 180,E1 -15686.731,E2 -15686.731} C_VEL
LIN {X 0,Y 312.506,Z 375.171,A -85,B 0,C 180,E1 -15689.655,E2 -15689.655} C_VEL
LIN {X 0,Y 312.522,Z 375.182,A -85,B 0,C 180,E1 -15693.689,E2 -15693.689} C_VEL
LIN {X 0,Y 312.513,Z 375.184,A -85,B 0,C 180,E1 -15697.388,E2 -15697.388} C_VEL
LIN {X 0,Y 312.474,Z 375.223,A -85,B 0,C 180,E1 -15698.9,E2 -15698.9} C_VEL
LIN {X 0,Y 312.912,Z 376.916,A -85,B 0,C 180,E1 -15699.458,E2 -15699.458} C_VEL
LIN {X 0,Y 315.808,Z 381.172,A -85,B 0,C 180,E1 -15700.109,E2 -15700.109} C_VEL
LIN {X 0,Y 322.49,Z 391.683,A -85,B 0,C 180,E1 -15701.56,E2 -15701.56} C_VEL
LIN {X 0,Y 330.142,Z 404.531,A -85,B 0,C 180,E1 -15703.13,E2 -15703.13} C_VEL
LIN {X 0,Y 338.775,Z 420.89,A -85,B 0,C 180,E1 -15704.822,E2 -15704.822} C_VEL
LIN {X 0,Y 342.447,Z 428.678,A -85,B 0,C 180,E1 -15705.526,E2 -15705.526} C_VEL
LIN {X 0,Y 338.46,Z 528.009,A -85,B 0,C 180,E1 -15707.608,E2 -15707.608} C_VEL
LIN {X 0,Y 337.692,Z 545.351,A -85,B 0,C 180,E1 -15708.067,E2 -15708.067} C_VEL
LIN {X 0,Y 336.409,Z 560.129,A -85,B 0,C 180,E1 -15708.666,E2 -15708.666} C_VEL
LIN {X 0,Y 334.751,Z 574.644,A -85,B 0,C 180,E1 -15709.494,E2 -15709.494} C_VEL
LIN {X 0,Y 332.65,Z 588.08,A -85,B 0,C 180,E1 -15710.472,E2 -15710.472} C_VEL
LIN {X 0,Y 330.474,Z 601.44,A -85,B 0,C 180,E1 -15711.729,E2 -15711.729} C_VEL
LIN {X 0,Y 327.939,Z 613.757,A -85,B 0,C 180,E1 -15713.126,E2 -15713.126} C_VEL
LIN {X 0,Y 325.306,Z 625.408,A -85,B 0,C 180,E1 -15714.734,E2 -15714.734} C_VEL
LIN {X 0,Y 322.522,Z 636.665,A -85,B 0,C 180,E1 -15716.618,E2 -15716.618} C_VEL
LIN {X 0,Y 319.904,Z 647.092,A -85,B 0,C 180,E1 -15718.754,E2 -15718.754} C_VEL
LIN {X 0,Y 317.602,Z 655.627,A -85,B 0,C 180,E1 -15720.868,E2 -15720.868} C_VEL
LIN {X 0,Y 315.849,Z 662.363,A -85,B 0,C 180,E1 -15722.881,E2 -15722.881} C_VEL
LIN {X 0,Y 313.956,Z 669.654,A -85,B 0,C 180,E1 -15725.536,E2 -15725.536} C_VEL
LIN {X 0,Y 312.554,Z 675.389,A -85,B 0,C 180,E1 -15728.222,E2 -15728.222} C_VEL
LIN {X 0,Y 311.814,Z 678.775,A -85,B 0,C 180,E1 -15730.24,E2 -15730.24} C_VEL
LIN {X 0,Y 311.138,Z 682.058,A -85,B 0,C 180,E1 -15732.924,E2 -15732.924} C_VEL
LIN {X 0,Y 310.789,Z 684.085,A -85,B 0,C 180,E1 -15735.597,E2 -15735.597} C_VEL
LIN {X 0,Y 310.626,Z 684.925,A -85,B 0,C 180,E1 -15738.251,E2 -15738.251} C_VEL
LIN {X 0,Y 310.513,Z 684.616,A -85,B 0,C 180,E1 -15740.884,E2 -15740.884} C_VEL
LIN {X 0,Y 310.723,Z 683.16,A -85,B 0,C 180,E1 -15743.507,E2 -15743.507} C_VEL
LIN {X 0,Y 310.953,Z 680.543,A -85,B 0,C 180,E1 -15746.112,E2 -15746.112} C_VEL
LIN {X 0,Y 311.361,Z 676.674,A -85,B 0,C 180,E1 -15748.707,E2 -15748.707} C_VEL
LIN {X 0,Y 311.932,Z 671.527,A -85,B 0,C 180,E1 -15751.291,E2 -15751.291} C_VEL
LIN {X 0,Y 312.924,Z 664.965,A -85,B 0,C 180,E1 -15753.863,E2 -15753.863} C_VEL
LIN {X 0,Y 314.233,Z 657.889,A -85,B 0,C 180,E1 -15756.098,E2 -15756.098} C_VEL
LIN {X 0,Y 315.82,Z 649.405,A -85,B 0,C 180,E1 -15758.317,E2 -15758.317} C_VEL
LIN {X 0,Y 317.696,Z 639.225,A -85,B 0,C 180,E1 -15760.516,E2 -15760.516} C_VEL
LIN {X 0,Y 319.688,Z 628.801,A -85,B 0,C 180,E1 -15762.377,E2 -15762.377} C_VEL
LIN {X 0,Y 321.632,Z 617.496,A -85,B 0,C 180,E1 -15764.069,E2 -15764.069} C_VEL
LIN {X 0,Y 323.619,Z 605.228,A -85,B 0,C 180,E1 -15765.59,E2 -15765.59} C_VEL
LIN {X 0,Y 325.563,Z 591.823,A -85,B 0,C 180,E1 -15766.944,E2 -15766.944} C_VEL
LIN {X 0,Y 327.271,Z 577.95,A -85,B 0,C 180,E1 -15768.062,E2 -15768.062} C_VEL
LIN {X 0,Y 328.648,Z 563.728,A -85,B 0,C 180,E1 -15768.952,E2 -15768.952} C_VEL
LIN {X 0,Y 329.819,Z 548.381,A -85,B 0,C 180,E1 -15769.65,E2 -15769.65} C_VEL
LIN {X 0,Y 330.598,Z 532.623,A -85,B 0,C 180,E1 -15770.11,E2 -15770.11} C_VEL
LIN {X 0,Y 333.947,Z 422.972,A -85,B 0,C 180,E1 -15772.446,E2 -15772.446} C_VEL
LIN {X 0,Y 333.22,Z 420.286,A -85,B 0,C 180,E1 -15772.581,E2 -15772.581} C_VEL
LIN {X 0,Y 324.548,Z 399.966,A -85,B 0,C 180,E1 -15773.953,E2 -15773.953} C_VEL
LIN {X 0,Y 319.8,Z 389.81,A -85,B 0,C 180,E1 -15774.717,E2 -15774.717} C_VEL
LIN {X 0,Y 317.441,Z 387.084,A -85,B 0,C 180,E1 -15775.047,E2 -15775.047} C_VEL
LIN {X 0,Y 307.769,Z 380.622,A -85,B 0,C 180,E1 -15776.333,E2 -15776.333} C_VEL
LIN {X 0,Y 305.851,Z 377.64,A -85,B 0,C 180,E1 -15776.647,E2 -15776.647} C_VEL
LIN {X 0,Y 305.451,Z 376.062,A -85,B 0,C 180,E1 -15776.78,E2 -15776.78} C_VEL
LIN {X 0,Y 305.435,Z 376.06,A -85,B 0,C 180,E1 -15780.412,E2 -15780.412} C_VEL
LIN {X 0,Y 305.469,Z 376.061,A -85,B 0,C 180,E1 -15784.078,E2 -15784.078} C_VEL
LIN {X 0,Y 305.457,Z 376.05,A -85,B 0,C 180,E1 -15786.742,E2 -15786.742} C_VEL
LIN {X 0,Y 305.413,Z 376.05,A -85,B 0,C 180,E1 -15790.589,E2 -15790.589} C_VEL
LIN {X 0,Y 305.425,Z 376.064,A -85,B 0,C 180,E1 -15793.655,E2 -15793.655} C_VEL
LIN {X 0,Y 305.439,Z 376.052,A -85,B 0,C 180,E1 -15797.418,E2 -15797.418} C_VEL
LIN {X 0,Y 305.444,Z 376.055,A -85,B 0,C 180,E1 -15801.592,E2 -15801.592} C_VEL
LIN {X 0,Y 305.464,Z 376.057,A -85,B 0,C 180,E1 -15804.886,E2 -15804.886} C_VEL
LIN {X 0,Y 305.445,Z 376.064,A -85,B 0,C 180,E1 -15808.358,E2 -15808.358} C_VEL
LIN {X 0,Y 305.477,Z 376.037,A -85,B 0,C 180,E1 -15811.109,E2 -15811.109} C_VEL
LIN {X 0,Y 305.481,Z 376.005,A -85,B 0,C 180,E1 -15814.079,E2 -15814.079} C_VEL
LIN {X 0,Y 305.47,Z 376.057,A -85,B 0,C 180,E1 -15818.4,E2 -15818.4} C_VEL
LIN {X 0,Y 305.546,Z 376.041,A -85,B 0,C 180,E1 -15821.214,E2 -15821.214} C_VEL
LIN {X 0,Y 305.63,Z 376.038,A -85,B 0,C 180,E1 -15825.347,E2 -15825.347} C_VEL
LIN {X 0,Y 305.627,Z 376.023,A -85,B 0,C 180,E1 -15829.399,E2 -15829.399} C_VEL
LIN {X 0,Y 305.748,Z 376.021,A -85,B 0,C 180,E1 -15832.072,E2 -15832.072} C_VEL
LIN {X 0,Y 305.66,Z 376.017,A -85,B 0,C 180,E1 -15834.722,E2 -15834.722} C_VEL
LIN {X 0,Y 305.949,Z 375.997,A -85,B 0,C 180,E1 -15838.683,E2 -15838.683} C_VEL
LIN {X 0,Y 305.941,Z 375.984,A -85,B 0,C 180,E1 -15841.316,E2 -15841.316} C_VEL
LIN {X 0,Y 305.666,Z 376.036,A -85,B 0,C 180,E1 -15845.276,E2 -15845.276} C_VEL
LIN {X 0,Y 305.748,Z 376.013,A -85,B 0,C 180,E1 -15847.927,E2 -15847.927} C_VEL
LIN {X 0,Y 305.597,Z 376.034,A -85,B 0,C 180,E1 -15851.945,E2 -15851.945} C_VEL
LIN {X 0,Y 305.56,Z 376.042,A -85,B 0,C 180,E1 -15854.979,E2 -15854.979} C_VEL
LIN {X 0,Y 305.556,Z 376.039,A -85,B 0,C 180,E1 -15858.784,E2 -15858.784} C_VEL
LIN {X 0,Y 305.487,Z 376.048,A -85,B 0,C 180,E1 -15863.039,E2 -15863.039} C_VEL
LIN {X 0,Y 305.47,Z 376.051,A -85,B 0,C 180,E1 -15866.197,E2 -15866.197} C_VEL
LIN {X 0,Y 305.449,Z 376.061,A -85,B 0,C 180,E1 -15869.033,E2 -15869.033} C_VEL
LIN {X 0,Y 305.436,Z 376.062,A -85,B 0,C 180,E1 -15871.952,E2 -15871.952} C_VEL
LIN {X 0,Y 305.461,Z 376.06,A -85,B 0,C 180,E1 -15875.113,E2 -15875.113} C_VEL
LIN {X 0,Y 305.41,Z 376.057,A -85,B 0,C 180,E1 -15878.519,E2 -15878.519} C_VEL
LIN {X 0,Y 305.434,Z 376.061,A -85,B 0,C 180,E1 -15882.581,E2 -15882.581} C_VEL
LIN {X 0,Y 305.42,Z 376.067,A -85,B 0,C 180,E1 -15886.344,E2 -15886.344} C_VEL
LIN {X 0,Y 305.421,Z 376.115,A -85,B 0,C 180,E1 -15889.453,E2 -15889.453} C_VEL
LIN {X 0,Y 308.38,Z 386.628,A -85,B 0,C 180,E1 -15892.522,E2 -15892.522} C_VEL
LIN {X 0,Y 309.555,Z 391.186,A -85,B 0,C 180,E1 -15893.762,E2 -15893.762} C_VEL
LIN {X 0,Y 319.831,Z 414.055,A -85,B 0,C 180,E1 -15895.508,E2 -15895.508} C_VEL
LIN {X 0,Y 324.231,Z 425.038,A -85,B 0,C 180,E1 -15896.244,E2 -15896.244} C_VEL
LIN {X 0,Y 327.229,Z 443.471,A -85,B 0,C 180,E1 -15897.003,E2 -15897.003} C_VEL
LIN {X 0,Y 323.679,Z 557.171,A -85,B 0,C 180,E1 -15899.5,E2 -15899.5} C_VEL
LIN {X 0,Y 322.555,Z 572.851,A -85,B 0,C 180,E1 -15900.06,E2 -15900.06} C_VEL
LIN {X 0,Y 320.989,Z 587.91,A -85,B 0,C 180,E1 -15900.846,E2 -15900.846} C_VEL
LIN {X 0,Y 319.16,Z 602.92,A -85,B 0,C 180,E1 -15901.912,E2 -15901.912} C_VEL
LIN {X 0,Y 317.113,Z 616.598,A -85,B 0,C 180,E1 -15903.156,E2 -15903.156} C_VEL
LIN {X 0,Y 315.084,Z 629.117,A -85,B 0,C 180,E1 -15904.572,E2 -15904.572} C_VEL
LIN {X 0,Y 312.733,Z 641.831,A -85,B 0,C 180,E1 -15906.315,E2 -15906.315} C_VEL
LIN {X 0,Y 310.769,Z 652.754,A -85,B 0,C 180,E1 -15908.143,E2 -15908.143} C_VEL
LIN {X 0,Y 309.001,Z 662.329,A -85,B 0,C 180,E1 -15910.052,E2 -15910.052} C_VEL
LIN {X 0,Y 307.178,Z 671.972,A -85,B 0,C 180,E1 -15912.353,E2 -15912.353} C_VEL
LIN {X 0,Y 305.677,Z 680.799,A -85,B 0,C 180,E1 -15914.937,E2 -15914.937} C_VEL
LIN {X 0,Y 304.742,Z 687.463,A -85,B 0,C 180,E1 -15917.344,E2 -15917.344} C_VEL
LIN {X 0,Y 304.027,Z 693.365,A -85,B 0,C 180,E1 -15920.016,E2 -15920.016} C_VEL
LIN {X 0,Y 303.796,Z 696.872,A -85,B 0,C 180,E1 -15922.021,E2 -15922.021} C_VEL
LIN {X 0,Y 303.615,Z 700.379,A -85,B 0,C 180,E1 -15924.687,E2 -15924.687} C_VEL
LIN {X 0,Y 303.616,Z 702.656,A -85,B 0,C 180,E1 -15927.346,E2 -15927.346} C_VEL
LIN {X 0,Y 303.618,Z 703.758,A -85,B 0,C 180,E1 -15930,E2 -15930} C_VEL
LIN {X 0,Y 303.602,Z 703.701,A -85,B 0,C 180,E1 -15932.654,E2 -15932.654} C_VEL
LIN {X 0,Y 303.586,Z 702.349,A -85,B 0,C 180,E1 -15935.473,E2 -15935.473} C_VEL
LIN {X 0,Y 303.775,Z 700.055,A -85,B 0,C 180,E1 -15937.979,E2 -15937.979} C_VEL
LIN {X 0,Y 304.26,Z 696.481,A -85,B 0,C 180,E1 -15940.649,E2 -15940.649} C_VEL
LIN {X 0,Y 305.226,Z 691.643,A -85,B 0,C 180,E1 -15943.312,E2 -15943.312} C_VEL
LIN {X 0,Y 306.564,Z 685.417,A -85,B 0,C 180,E1 -15945.968,E2 -15945.968} C_VEL
LIN {X 0,Y 308.555,Z 677.639,A -85,B 0,C 180,E1 -15948.595,E2 -15948.595} C_VEL
LIN {X 0,Y 310.748,Z 669.398,A -85,B 0,C 180,E1 -15950.868,E2 -15950.868} C_VEL
LIN {X 0,Y 313.336,Z 659.416,A -85,B 0,C 180,E1 -15953.131,E2 -15953.131} C_VEL
LIN {X 0,Y 316.469,Z 647.548,A -85,B 0,C 180,E1 -15955.309,E2 -15955.309} C_VEL
LIN {X 0,Y 319.242,Z 636.336,A -85,B 0,C 180,E1 -15957.004,E2 -15957.004} C_VEL
LIN {X 0,Y 322.343,Z 622.819,A -85,B 0,C 180,E1 -15958.663,E2 -15958.663} C_VEL
LIN {X 0,Y 325.028,Z 609.422,A -85,B 0,C 180,E1 -15959.991,E2 -15959.991} C_VEL
LIN {X 0,Y 327.471,Z 595.371,A -85,B 0,C 180,E1 -15961.092,E2 -15961.092} C_VEL
LIN {X 0,Y 329.49,Z 581.07,A -85,B 0,C 180,E1 -15961.955,E2 -15961.955} C_VEL
LIN {X 0,Y 331.206,Z 565.615,A -85,B 0,C 180,E1 -15962.623,E2 -15962.623} C_VEL
LIN {X 0,Y 332.249,Z 550.557,A -85,B 0,C 180,E1 -15963.048,E2 -15963.048} C_VEL
LIN {X 0,Y 336.246,Z 445.627,A -85,B 0,C 180,E1 -15965.327,E2 -15965.327} C_VEL
LIN {X 0,Y 334.452,Z 435.901,A -85,B 0,C 180,E1 -15965.84,E2 -15965.84} C_VEL
LIN {X 0,Y 326.812,Z 419.884,A -85,B 0,C 180,E1 -15967.405,E2 -15967.405} C_VEL
LIN {X 0,Y 320.55,Z 408.203,A -85,B 0,C 180,E1 -15968.733,E2 -15968.733} C_VEL
LIN {X 0,Y 315.34,Z 399.087,A -85,B 0,C 180,E1 -15969.886,E2 -15969.886} C_VEL
